(* CODESYS project IoDrvMasterTemplateIEC.library
   Author: 3S - Smart Software Solutions GmbH
   Title: IoDrvMasterTemplateIEC
   Version: 3.5.15.0
   Placeholder: PlaceholderTemplate
   DocFormat: reStructuredText
   Company: MyCompany
   LanguageModelAttribute: qualified-access-only
   DefaultNamespace: TMP

Project tree, tasks and I/O mapping:
  libraries: SysMem, * (System); SysCpuHandling, * (System); IoDrvBase, * (System); IoDriver Parameter Interfaces, * (System); Base Interfaces, * (System); IoDriver Interfaces, * (System); CmpErrors2 Interfaces, * (System); SysTypes2 Interfaces, * (System); CAA Device Diagnosis, * (CAA Technical Workgroup); CAA Types Extern, * (CAA Technical Workgroup); CmpAsyncMgr, * (System); Network, 3.5.7.0 (3S - Smart Software Solutions GmbH); IoStandard, 3.5.13.0 (System); IoDrvUtility, 3.5.15.0 (3S - Smart Software Solutions GmbH); SysSem, * (System)
  00000000-0000-0000-0000-000000000000|D:\CoDeSys\LibrariesV3\trunk\Intern\CAA\CAA Template\3.2.0.3 draft\Prefix.pdf
  00000000-0000-0000-0000-000000000000|D:\CoDeSys\LibrariesV3\trunk\Intern\CAA\CAA Template\3.4.0.0 draft\Placeholder.xml
  00000000-0000-0000-0000-000000000000|D:\CoDeSys\LibrariesV3\trunk\Intern\CAA\CAA Template\3.5.2.0 draft\Placeholder.xml
  IoDrvMasterTemplateIEC/
    Enums/
      data type IoType
    Function Blocks/
      function block FixedArrayList [ST]: Create, Destroy, Get, Size
      function block IoDrvTemplateMaster [ST]: IoDrvReadInputs, IoDrvIdentify, IoDrvUpdateConfiguration, IoDrvWatchdogTrigger, IoDrvScanModules, IoDrvUpdateMapping, IoDrvWriteOutputs, IoDrvStartBusCycle, IoDrvGetModuleDiagnosis, IoDrvWriteParameter, IoDrvReadParameter, QueryInterface, FB_Reinit, Initialize, FB_Exit, FB_Init, IoDrvGetConnector, Cleanup, FreeScanData
      function block IoDrvTemplateModule [ST]: Initialize, UpdateConfigurationCreate, UpdateConfigurationDestroy, StartBusCycle, ModuleID, IsDisabled
      function block IoDrvTemplateSlave [ST]: Initialize, UpdateConfigurationCreate, UpdateConfigurationDestroy, StartBusCycle, SlaveID, IsDisabled
      function block IoDrvTemplateMasterDiag [ST]: ChildNodeCount, Connector, Enable, FirstChildNode, Index, IsRootNode, NextSiblingNode, ParentNode, SiblingNodeCount, GetChild, Initialize_Diag, GetSpecificDeviceState, SetCommunicationState, GetDeviceInfo, GetDeviceErrorAsync, GetSpecificDeviceErrorAsync, GetDeviceDiagnosisInfo, GetDeviceState, CheckCurrentSupportedCommunicationState, CheckSupportedCommunicationState, GetQoS, GetBusErrorAsync, GetBusDiagnosisInfo, GetBusState, GetBusInfo, GetSpecificBusState, GetLogger, GetBusScanAsync, ReconfigureActive, SiblingIRP, ReconfigureAsync, RegisterIRPChild
      function block IoDrvTemplateSlaveDiag [ST]: ChildNodeCount, Connector, Enable, FirstChildNode, Index, IsRootNode, NextSiblingNode, ParentNode, SiblingNodeCount, GetChild, Initialize_Diag, GetSpecificDeviceState, SetCommunicationState, GetDeviceInfo, GetDeviceErrorAsync, GetSpecificDeviceErrorAsync, GetDeviceDiagnosisInfo, GetDeviceState, CheckCurrentSupportedCommunicationState, CheckSupportedCommunicationState, GetQoS, GetBusErrorAsync, GetBusDiagnosisInfo, GetBusState, GetBusInfo, GetSpecificBusState
      function block IoDrvTemplateModuleDiag [ST]: ChildNodeCount, Connector, Enable, FirstChildNode, Index, IsRootNode, NextSiblingNode, ParentNode, SiblingNodeCount, GetChild, Initialize_Diag, GetSpecificDeviceState, SetCommunicationState, GetDeviceInfo, GetDeviceErrorAsync, GetSpecificDeviceErrorAsync, GetDeviceDiagnosisInfo, GetDeviceState, CheckCurrentSupportedCommunicationState, CheckSupportedCommunicationState, GetQoS, GetBusErrorAsync, GetBusDiagnosisInfo, GetBusState, GetBusInfo, GetSpecificBusState
    GlobalConstants/
      global variables PARAMS_IODRVTEMPLATEMASTER
    Structs/
      data type IoEntry
      data type Module
      data type Slave
      data type UdpIO
    _ExternalFilesDoku/
      M_AblaufProto
      M_Behave
      M_Connectors
      M_cycle
      M_Proto
      M_Tree
      M_run
  00000000-0000-0000-0000-000000000000|D:\CODESYS\CodesysSpV3\CodesysSpV3\Templates\IoDrvMasterTemplateIEC\RestoreOld\DokPic\M_AblaufProto.png
  00000000-0000-0000-0000-000000000000|D:\CODESYS\CodesysSpV3\CodesysSpV3\Templates\IoDrvMasterTemplateIEC\RestoreOld\DokPic\M_Behave.png
  00000000-0000-0000-0000-000000000000|D:\CODESYS\CodesysSpV3\CodesysSpV3\Templates\IoDrvMasterTemplateIEC\RestoreOld\DokPic\M_Connectors.png
  00000000-0000-0000-0000-000000000000|D:\CODESYS\CodesysSpV3\CodesysSpV3\Templates\IoDrvMasterTemplateIEC\RestoreOld\DokPic\M_cycle.png
  00000000-0000-0000-0000-000000000000|D:\CODESYS\CodesysSpV3\CodesysSpV3\Templates\IoDrvMasterTemplateIEC\RestoreOld\DokPic\M_Proto.png
  00000000-0000-0000-0000-000000000000|D:\CODESYS\CodesysSpV3\CodesysSpV3\Templates\IoDrvMasterTemplateIEC\RestoreOld\DokPic\M_Tree.png
  00000000-0000-0000-0000-000000000000|D:\CODESYS\CodesysSpV3\CodesysSpV3\Templates\IoDrvMasterTemplateIEC\RestoreOld\DokPic\M_run.png
*)

// IoDrvMasterTemplateIEC/Structs/IoEntry
/// Is generated for each output and input, when an ouput or input exsits in the Slave (type 3) or modules(all types).
/// This saves time in ``IoDrvTemplateMaster.IoDrvStartBusCycle``, because iterating over the ConnectorList and searching for the out- and inputs takes time. This is done in ''IoDrvTemplateMaster.IoDrvUpdateConfiguration'', where a fixed arrayList is generated. 
TYPE IoEntry :
STRUCT
    /// Input or output?
	ioType: IoType;
    /// Pointer to the Parameter. 
	pParameter: POINTER TO IoConfigParameter;
END_STRUCT
END_TYPE

// IoDrvMasterTemplateIEC/Structs/Module
/// This struct is generated, for each Module in the device tree in the ''IoDrvTemplateSlave'' FB, to access the Slaves over a pointer an not over the ConenctorList. This saves time in the ''IoDrvTemplateMaster.IoDrvStartBusCycle'' method. 
TYPE Module :
STRUCT
	moduleInstance : POINTER TO IoDrvTemplateModule;		
END_STRUCT
END_TYPE

// IoDrvMasterTemplateIEC/Structs/Slave
/// This struct is generated, for each Slave in the device tree in the ''IoDrvTemplateMaster'' FB, to access the Slaves over a pointer an not over the ConenctorList. This saves time in the ''IoDrvTemplateMaster.IoDrvStartBusCycle'' method. 
TYPE Slave :
STRUCT
	slaveInstance : POINTER TO IoDrvTemplateSlave;		
END_STRUCT
END_TYPE

// IoDrvMasterTemplateIEC/Structs/UdpIO
/// Information, which are needed also in the modules an slaves. This struct function is to bundle this information and pass them down in the stack easily. 
TYPE UdpIO :
STRUCT
	r_udpInBuffer: POINTER TO FixedArrayList;
	r_BytesReceived : CAA.SIZE;

	s_udpSender : POINTER TO NBS.UDP_Send;
	s_udpPeer: POINTER TO NBS.UDP_Peer ;
	s_portSendTo : UINT;
	s_ipSendTo : POINTER TO NBS.IP_ADDR;
	s_udpOutBuffer: POINTER TO FixedArrayList;	
END_STRUCT
END_TYPE

// IoDrvMasterTemplateIEC/Enums/IoType
{attribute 'qualified_only'}
{attribute 'strict'}
/// Used in |IoEntry|.
TYPE IoType :
(
	INPUT := 0,
	OUTPUT := 1
);
END_TYPE

// IoDrvMasterTemplateIEC/GlobalConstants/PARAMS_IODRVTEMPLATEMASTER
VAR_GLOBAL
	/// This string is used, when memory is allocated. 
    g_stComponentName : STRING := 'IoDrvMasterTemplate';
	
	/// The ID at which the ParameterId for the inputs start in the deviceDescription (xml-file). This is a running nummer. The loop stops, if there is an unused number: 2000, 2001, 2002, 2004 --> after 2002 no entries would be processed.
	START_OF_INPUTPARAMS : UDINT := 2000;
   
	/// The ID at which the ParameterId for the inputs end in the deviceDescription (xml-file).
	END_OF_INPUTPARAMS : UDINT := 2999;

    /// Same as for inputs. 	
	START_OF_OUTPUTPARAMS : UDINT := 3000;
    /// Same as for inputs. 
	END_OF_OUTPUTPARAMS : UDINT := 3999;

    /// The size of the UDP-Buffer to send messages.  
	SIZE_OF_INPUT_OUTPUT_BUFFER : UDINT := 30;
	
END_VAR

// IoDrvMasterTemplateIEC/Function Blocks/FixedArrayList
(*
 .. code-block:: codesys
  
    VAR_GLOBAL CONSTANT
        g_stComponentName : STRING := 'MyApp';
    END_VAR
    
    TYPE MyStruct:
    STRUCT
        someData1: DWORD;
        someData2: BYTE;
    END_STRUCT
    END_TYPE
    
    _fixedArrayList :FixedArrayList
    pMyStruct : POINTER TO MyStruct;
    numberOfEntries: DWORD;
    
    numberOfEntries := 10;
    IF( NOT _fixedArrayList(numberOfEntries, SIZEOF(MyStruct:), g_stComponentName) ) THEN 
        RETURN; //error no free space ....
    END_IF
    
	IF _fixedArrayList.Size > 0 THEN
		FOR i:=0 TO _fixedArrayList.Size - 1 DO
			pMyStruct := _fixedArrayList.Get(i);
			// do something ...			
		END_FOR
	END_IF
*)
FUNCTION_BLOCK FixedArrayList
VAR_INPUT
END_VAR
VAR_OUTPUT
END_VAR
VAR
    /// Address to the memblock. 
	_varMem: POINTER TO BYTE := 0;
    /// How many entries.
	_sizeOfArray: DWORD;
    /// Given in Create.
	_sizeOfObjectInByte: DWORD;
    /// Needed by Destroy
	_stComponentName: STRING;
END_VAR

/// Creates a fixed memmory block, which can be accessed over an index.
METHOD Create : BOOL
VAR_INPUT
    /// How many entries should be available?
	sizeOfArray: DWORD;
    /// How big in bytes is one entry?
	sizeOfObjectInByte: DWORD;
    /// Which component is using this memory? If the memory is not freed after shutdown, a warning with this string is generated.
	stComponentName : STRING;
END_VAR

VAR
	iecResult : RTS_IEC_Result;
END_VAR
_sizeOfArray := sizeOfArray;
_sizeOfObjectInByte := sizeOfObjectInByte;
_stComponentName := stComponentName;
_varMem :=  SysMemAllocData(_stComponentName, _sizeOfObjectInByte*_sizeOfArray , ADR(iecResult));


Create := (iecResult = CmpErrors.Errors.ERR_OK); // if false -> _varMem=0 (impicit)
END_METHOD

/// Frees the memory, which was allocated in |FixedArrayList.Create|, if it was successful.
METHOD Destroy
VAR_INPUT
END_VAR
IF(_varMem <> 0) THEN
	SysMemFreeData(_stComponentName, _varMem);
END_IF
END_METHOD

/// Returns a pointer to the element at the given index.
/// :return: The address to the element, if the index is valid, else 0.
METHOD Get : POINTER TO BYTE
VAR_INPUT
    /// Index of the element, which should be accessed. The index is between 0 and DWORD.maxValue.
	index: DWORD;
END_VAR
IF( index < _sizeOfArray) THEN
	Get := (_varMem + _sizeOfObjectInByte*index);
ELSE
	Get := 0;
END_IF
END_METHOD

/// Reads the amount of elements, which can be accessed. Is for the use in loops to iterate over all elements. 
PROPERTY Size : DWORD
GET
Size := _sizeOfArray;
END_GET
END_PROPERTY

END_FUNCTION_BLOCK

// IoDrvMasterTemplateIEC/Function Blocks/IoDrvTemplateMaster
{attribute 'no_assign'}
{attribute 'conditionalshow_all_locals' := 'IoDrvDebug'}
FUNCTION_BLOCK IoDrvTemplateMaster EXTENDS IoDrvBase IMPLEMENTS ICmpIoDrvParameter
VAR_INPUT
END_VAR
VAR_OUTPUT
END_VAR
VAR CONSTANT
	CLASSID_CCmpIoDrvTemplate : DWORD := 16#0000FF02;
END_VAR
VAR
	_IIoDrv : ICmpIoDrv;
	_IIoDrvParameter : ICmpIoDrvParameter;
	
	_xBackGroundDiagStarted : BOOL;
	_bDeactivated : BOOL;

    // used to save the slaves with their slaveID in a list. To access the correct slave in the method IoDrvStartBusCylce fast.  
	_fal_shortcut2Slaves :FixedArrayList; 
	
	//Variables for scan
	_iScannedSlaves : INT;
	_pScanList : POINTER TO IoStandard.IoConfigConnector;

    // UDP server varaibles
	_udpPeer: NBS.UDP_Peer ;
	_iPAddr :  NBS.IP_ADDR;
	_uiPortReceive : UINT;
	_udpRec : NBS.UDP_Receive;
	_udpSend : NBS.UDP_Send;
	_udpInBuffer, _udpOutBuffer: FixedArrayList;

	_myState: BYTE := 1; // remember the state
	_connectorFlagController: IoDrvUtility.ConnectorFlagController;
	
//	_lock: RTS_IEC_Handle;
END_VAR

{attribute 'conditionalshow' := 'IoDrvDebug'}
METHOD IoDrvReadInputs : UDINT
VAR_INPUT
	pConnectorMapList : POINTER TO IoConfigConnectorMap;
	nCount : DINT;
END_VAR
VAR
	i,j : DINT;
	pConnectorMap : POINTER TO IoStandard.IoConfigConnectorMap;
	pChannelMap : POINTER TO IoStandard.IoConfigChannelMap;
END_VAR
IoDrvReadInputs_Count := IoDrvReadInputs_Count + 1;

IF pConnectorMapList = 0 OR nCount = 0 THEN
	IoDrvReadInputs := Errors.ERR_PARAMETER;
	RETURN;
END_IF

FOR i:=0 TO nCount - 1 DO
	pConnectorMap := ADR(pConnectorMapList[i]);
	
	FOR j:= 0 TO UDINT_TO_UINT(pConnectorMap^.dwNumOfChannels) - 1 DO
		pChannelMap := ADR(pConnectorMap^.pChannelMapList[j]);
		
		// input medium byteorder: Little Endian:		
		IoMgrCopyInputLE(pChannelMap, pChannelMap^.pParameter^.dwDriverSpecific);
		
		// input medium byteorder: Big Endian:		
		//IoMgrCopyInputBE(ADR(pChannelMap, pChannelMap^.pParameter^.dwDriverSpecific);
	END_FOR
END_FOR

IoDrvReadInputs := Errors.ERR_OK;
END_METHOD

{attribute 'conditionalshow' := 'IoDrvDebug'}
METHOD IoDrvIdentify : UDINT
VAR_INPUT
	pConnector : POINTER TO IoConfigConnector;	
END_VAR
VAR
END_VAR
IoDrvIdentify_Count := IoDrvIdentify_Count + 1;
IoDrvIdentify := Errors.ERR_NOTIMPLEMENTED;
END_METHOD

{attribute 'conditionalshow' := 'IoDrvDebug'}
METHOD IoDrvUpdateConfiguration : UDINT
VAR_INPUT
	pConnectorList : POINTER TO IoConfigConnector;
	nCount : DINT;
END_VAR
VAR
	p_dwParValueSlave : POINTER TO IoDrvTemplateSlave;
	pParameter : POINTER TO IoConfigParameter;	
	pDummy			: POINTER TO XWORD;
	
	pChild : POINTER TO IoConfigConnector;	
	pstConnectorVendorName : POINTER TO STRING;
	pstConnectorDeviceName : POINTER TO STRING;
	dwTest,i : DWORD;
	Result : UDINT := 0;
	xDisabled : BOOL;
	
	slaveCount : UDINT := 0;
	slaveIter : POINTER TO Slave;
	
	nCountRemember: DINT;
	
	pstDummy : POINTER TO STRING;
END_VAR
IoDrvUpdateConfiguration_Count := IoDrvUpdateConfiguration_Count + 1;
IoDrvUpdateConfiguration := Errors.ERR_OK;

IF pConnectorList = 0 THEN // destroy -> time to clean up
	// Reset application
	m_pConnector^.hIoDrv := 0; 
	m_pConnector^.pFather^.hIoDrv := 0;
	
	Cleanup();
	_udpOutBuffer.Destroy();
	_udpInBuffer.Destroy();
	//Go through all childs of the device
	IF _fal_shortcut2Slaves.Size > 0 THEN
		FOR i:=0 TO _fal_shortcut2Slaves.Size - 1 DO
			slaveIter := _fal_shortcut2Slaves.Get(i);
			slaveIter^.slaveInstance^.UpdateConfigurationDestroy(); // childs of master are IoDrvTemplateSlave FB´s -> call UpdateConfigurationDestroy(...) to give them the chance to cleanup
		END_FOR
	END_IF
	_fal_shortcut2Slaves.Destroy();// delete shortcut list to slaves 	

	// reset var´s (needed when reconfigure is activated)
	_iScannedSlaves := 0;
	_pScanList := 0;
	_myState := 1; // remember the state
	
	RETURN; // nothing more to do
END_IF

m_pConnector := IoMgrConfigGetConnector(pConnectorList, ADR(nCount), m_wModuleType, m_dwInstance);
nCountRemember := nCount; // to reset the counter to iterate over the childs
_connectorFlagController.Init(m_pConnector, nCount, FALSE); // ^.pFather is MasterIECDriver::Connector::256
_connectorFlagController.AutoSetErrorClearedFlag := TRUE; //use the generic algorithm for setting the Error Cleared flag in device tree.
_connectorFlagController.DiagProvider := TRUE;

IF m_pConnector = 0 THEN
	IoDrvUpdateConfiguration := ERRORS.ERR_PARAMETER;
	RETURN;
END_IF

//check if device is enabled in the device tree
_bDeactivated := _connectorFlagController.State = IoDrvUtility.ConnectorState.DISABLED;

IF _bDeactivated THEN // IO changes don´t care, if device is disabled.
	m_pConnector^.hIoDrv := 0;
	m_pConnector^.pFather^.hIoDrv := 0;
	IoDrvUpdateConfiguration := CmpErrors.Errors.ERR_OK;
	RETURN;
END_IF

IF (m_pConnector^.hIoDrv = 0) and (NOT _bDeactivated) THEN // register to get called, when IO changed
	m_pConnector^.hIoDrv := m_hInterface; 
	m_pConnector^.pFather^.hIoDrv := m_hInterface;
END_IF

IF m_pConnector^.hIoDrv = m_hInterface THEN
	{IF defined (pou:IoMgrSetDriverProperties)}			
		IoMgrSetDriverProperties(m_hInterface, DRVPROP_CONSISTENCY OR DRVPROP_BACKGROUND_GETDIAG);
		//Note: background diagnosis property flag is optional (supported with 3.5.1.0 runtime)
	{END_IF}										

	//Read some parameters
	pParameter := IoMgrConfigGetParameter(m_pConnector, 393218);
	IF pParameter <> 0 THEN
		pstConnectorVendorName := IoMgrConfigGetParameterValuePointer(pParameter, ADR(Result));
	END_IF
	pParameter := IoMgrConfigGetParameter(m_pConnector, 393219);
	IF pParameter <> 0 THEN
		pstConnectorDeviceName := IoMgrConfigGetParameterValuePointer(pParameter, ADR(Result));
	END_IF
	pParameter := IoMgrConfigGetParameter(m_pConnector, 393220);	(* test parameter *)
	IF (pParameter <> 0) THEN
		dwTest := IoMgrConfigGetParameterValueDword(pParameter, ADR(Result));	(* Test parameter value *)			
	END_IF
	
	pParameter := IoMgrConfigGetParameter(m_pConnector, 256);	// ip addr
	IF (pParameter <> 0) THEN
		pstDummy := IoMgrConfigGetParameterValuePointer(pParameter, ADR(Result));
		_iPAddr.sAddr := pstDummy^;
	END_IF
	
	pParameter := IoMgrConfigGetParameter(m_pConnector, 257);	// port
	IF (pParameter <> 0) THEN
		_uiPortReceive := DWORD_TO_UINT( IoMgrConfigGetParameterValueWord (pParameter, ADR(Result)) );		
	END_IF

	
	//Go through all childs of the device
	nCount:= nCountRemember;
	slaveCount :=0; // save amount of slaves
	pChild := IoMgrConfigGetFirstChild(m_pConnector, ADR(nCount), m_pConnector);
	WHILE (pChild <> 0) DO
		// childs of master are IoDrvTemplateSlave FB´s -> call UpdateConfigurationCreate(...) to let them init()
		pParameter := IoMgrConfigGetParameter(pChild, 1); 
		IF pParameter <> 0 THEN
			pDummy := ConfigGetParameterValuePointer(pParameter,ADR(Result));
			p_dwParValueSlave :=  pDummy^;
			IF p_dwParValueSlave <> 0 THEN
				p_dwParValueSlave^.UpdateConfigurationCreate(pConnector := pChild, m_hInterface, nCount, xDisabled => xDisabled);
				IF NOT xDisabled THEN
					slaveCount := slaveCount + 1;
				END_IF
			END_IF
		END_IF

		pChild := IoMgrConfigGetNextChild(pChild, ADR(nCount), m_pConnector);
	END_WHILE
	
	// save a shortcut to know which IoDrvTemplateSlave instance is in resposable to which slaveID and save this in a variable memory block (_fal_shortcut2Slaves) to access it without going over the slowly connectorList (IoMgrConfigGetFirstChild) 
	// this _fal_shortcut2Slaves is needed in the IoDrvStartBusCycle method to be fast
	IF( NOT _fal_shortcut2Slaves.Create( slaveCount, SIZEOF(Slave), g_stComponentName) ) THEN
		IoDrvUpdateConfiguration := Errors.ERR_FAILED; // no space ....
		RETURN;
	END_IF
	
	nCount:= nCountRemember;
	pChild := IoMgrConfigGetFirstChild(m_pConnector, ADR(nCount), m_pConnector);
	i := 0;
	WHILE (pChild <> 0) DO
		pParameter := IoMgrConfigGetParameter(pChild, 1); 
		IF pParameter <> 0 THEN
			pDummy := ConfigGetParameterValuePointer(pParameter,ADR(Result));
			p_dwParValueSlave :=  pDummy^;
			IF p_dwParValueSlave <> 0 THEN
				IF NOT p_dwParValueSlave^.IsDisabled THEN
					slaveIter := _fal_shortcut2Slaves.Get(i); // get next place to save the slaveInstance
					i := i + 1;
					slaveIter^.slaveInstance := p_dwParValueSlave;
				END_IF
			END_IF
		END_IF
		pChild := IoMgrConfigGetNextChild(pChild, ADR(nCount), m_pConnector);
	END_WHILE

	_connectorFlagController.State := IoDrvUtility.ConnectorState.RUNNING;
END_IF
END_METHOD

{attribute 'conditionalshow' := 'IoDrvDebug'}
METHOD IoDrvWatchdogTrigger : UDINT
VAR_INPUT
	pConnector : POINTER TO IoConfigConnector;	
END_VAR
VAR
END_VAR
IoDrvWatchdogTrigger_Count := IoDrvWatchdogTrigger_Count + 1;
IoDrvWatchdogTrigger := Errors.ERR_OK;
END_METHOD

{attribute 'conditionalshow' := 'IoDrvDebug'}
METHOD IoDrvScanModules : UDINT
VAR_INPUT
	pConnector : POINTER TO IoConfigConnector;
	ppConnectorList : POINTER TO POINTER TO IoConfigConnector;
	pnCount : POINTER TO DINT;	
END_VAR
VAR
	pCurConnector : POINTER TO IoConfigConnector;
	pParameter: POINTER TO IoConfigParameter;
	pString : POINTER TO STRING;
	i : INT;
END_VAR
IoDrvScanModules_Count := IoDrvScanModules_Count + 1;

IF pConnector = 0 OR ppConnectorList = 0 OR pnCount = 0 THEN
	IoDrvScanModules := Errors.ERR_PARAMETER;
	RETURN;
END_IF

FreeScanData();

pnCount^ := 0;
ppConnectorList^ := 0;

(*
	TODO: implement specific bus scan!
	Note: IoDrvScanModules is called in communication task. If this method takes too long (> 20s) a communication timeout may happen.
	In this cases you can do a segmented scan by setting IoStandard.ConnectorOptions.CO_SCAN_PENDING_SUPPORTED.
	If IoDrvScanModules returns ERR_PENDING method is called again. The results of all calls are combined by the GUI.
*)

(*The following code just generates some example data. The real scan algorithm has to set the values regarding to the scan result. *)
_iScannedSlaves := 2; //we return 2 slaves

IF _iScannedSlaves > 0 THEN
	//Allocate memory for the connector list
	ppConnectorList^ := SysMemAllocData(g_stComponentName, UINT_TO_DWORD(INT_TO_UINT(_iScannedSlaves) * SIZEOF(IoStandard.IoConfigConnector)), 0);
	IF ppConnectorList = 0 THEN
		IoDrvScanModules := Errors.ERR_FAILED;
		_iScannedSlaves := 0;
		RETURN;
	END_IF
	SysMem.SysMemSet(ppConnectorList^, 0, UINT_TO_DWORD(INT_TO_UINT(_iScannedSlaves) * SIZEOF(IoStandard.IoConfigConnector)));
END_IF

pCurConnector := ppConnectorList^;
FOR i := 0 TO _iScannedSlaves - 1 DO
	pCurConnector^.dwNumOfParameters := 4; //we return the 4 mandatory parameters
	//Alocate memory for the parameter list of the current connector
	pCurConnector^.pParameterList := SysMemAllocData(g_stComponentName, pCurConnector^.dwNumOfParameters * SIZEOF(IoStandard.IoConfigParameter), 0);
	SysMem.SysMemSet(pCurConnector^.pParameterList, 0, pCurConnector^.dwNumOfParameters * SIZEOF(IoStandard.IoConfigParameter));
	
    pParameter := pCurConnector^.pParameterList;
	
	//Set parameter: Vendor code
	pParameter^.dwParameterId := 1;
	pParameter^.dwValue := 1; //Vendor Code
	pParameter^.wLen := 32;
	pParameter^.wType := INT_TO_WORD(TypeClass.TYPE_DWORD); //16#4
	pParameter^.dwFlags := IoStandard.PVF_READ OR IoStandard.PVF_WRITE OR IoStandard.PVF_VALUE; //16#34
	
	pParameter := pParameter + SIZEOF(IoStandard.IoConfigParameter);
	
	//Set parameter: Product code
	pParameter^.dwParameterId := 2;
	pParameter^.dwValue := 2; //Product Code
	pParameter^.wLen := 32;
	pParameter^.wType := INT_TO_WORD(TypeClass.TYPE_DWORD); //16#4
	pParameter^.dwFlags := IoStandard.PVF_READ OR IoStandard.PVF_WRITE OR IoStandard.PVF_VALUE; //16#34
	
	pParameter := pParameter + SIZEOF(IoStandard.IoConfigParameter);
	
	//Set parameter: Revision Number
	pParameter^.dwParameterId := 3;
	pParameter^.dwValue :=3; //Revision Number
	pParameter^.wLen := 32;
	pParameter^.wType := INT_TO_WORD(TypeClass.TYPE_DWORD); //16#4
	pParameter^.dwFlags := IoStandard.PVF_READ OR IoStandard.PVF_WRITE OR IoStandard.PVF_VALUE; //16#34
	
	pParameter := pParameter + SIZEOF(IoStandard.IoConfigParameter);
	
	
	(* Slave_T1_IECDriver.xml:
	
			<DeviceIdentification>
				<Type>40102</Type>
				<Id>1001 0001</Id>
	*)		
			
	//Set parameter: Device Identification
	pParameter^.dwParameterId := 4;
	pParameter^.dwValue := SysMemAllocData(g_stComponentName, SIZEOF(STRING), 0);
	pString := pParameter^.dwValue;
	pString^ := '1001 0001'; // Device Identification <Id>1001 0001</Id>
	pParameter^.wLen := SIZEOF(STRING);
	pParameter^.wType := INT_TO_WORD(TypeClass.TYPE_STRING); //16#10
	pParameter^.dwFlags := IoStandard.PVF_READ OR IoStandard.PVF_WRITE OR IoStandard.PVF_POINTER; //16#32
		
	pCurConnector^.hIoDrv := THIS;
	pCurConnector^.pFather := pConnector;
	pCurConnector^.wType := 40102; // <Type>40102</Type>
	
	pCurConnector := pCurConnector + SIZEOF(IoStandard.IoConfigConnector);
END_FOR

pnCount^ := _iScannedSlaves; //Set number of scanned devices
IoDrvScanModules := CmpErrors.Errors.ERR_OK;
END_METHOD

{attribute 'conditionalshow' := 'IoDrvDebug'}
METHOD IoDrvUpdateMapping : UDINT
VAR_INPUT
	pTaskMapList : POINTER TO IoConfigTaskMap;
	nCount : DINT;	
END_VAR
VAR
END_VAR
IoDrvUpdateMapping_Count := IoDrvUpdateMapping_Count + 1;

IF (pTaskMapList = 0) THEN
	IoDrvUpdateMapping := Errors.ERR_PARAMETER;
	RETURN;
END_IF

IoDrvUpdateMapping := Errors.ERR_OK;
END_METHOD

{attribute 'conditionalshow' := 'IoDrvDebug'}
METHOD IoDrvWriteOutputs : UDINT
VAR_INPUT
	pConnectorMapList : POINTER TO IoConfigConnectorMap;
	nCount : DINT;
END_VAR
VAR
	i,j : DINT;
	pConnectorMap : POINTER TO IoStandard.IoConfigConnectorMap;
	pChannelMap : POINTER TO IoStandard.IoConfigChannelMap;
END_VAR
IoDrvWriteOutputs_Count := IoDrvWriteOutputs_Count + 1;

IF pConnectorMapList = 0 OR nCount = 0 THEN
	IoDrvWriteOutputs := Errors.ERR_PARAMETER;
	RETURN;
END_IF

FOR i:=0 TO nCount - 1 DO
	pConnectorMap := ADR(pConnectorMapList[i]);
	
	FOR j:= 0 TO UDINT_TO_UINT(pConnectorMap^.dwNumOfChannels) - 1 DO
		pChannelMap := ADR(pConnectorMap^.pChannelMapList[j]);
		
		// output medium byteorder: Little Endian:		
		IoMgrCopyOutputLE(pChannelMap, pChannelMap^.pParameter^.dwDriverSpecific);
		
		// output medium byteorder: Big Endian:		
		//IoMgrCopyOutputBE(pChannelMap, pChannelMap^.pParameter^.dwDriverSpecific);
	END_FOR
END_FOR

IoDrvWriteOutputs := Errors.ERR_OK;
END_METHOD

{attribute 'conditionalshow' := 'IoDrvDebug'}
METHOD IoDrvStartBusCycle : UDINT
VAR_INPUT
	pConnector : POINTER TO IoConfigConnector;
END_VAR
VAR
	i : DWORD;
	slaveIter : POINTER TO Slave;
	udpIo: UdpIO;
	ipMulti :  NBS.IP_ADDR;
END_VAR
IoDrvStartBusCycle_Count := IoDrvStartBusCycle_Count + 1;

IF _bDeactivated OR_ELSE pConnector <> m_pConnector THEN
	RETURN;
END_IF

//if background diagnosis is not active call IoDrvGetModuleDiagnosis; normally it will be called by the runtime if DRVPROP_BACKGROUND_GETDIAG is set
IF NOT _xBackGroundDiagStarted THEN
	IoDrvGetModuleDiagnosis(m_pConnector); //DRVPROP_BACKGROUND_GETDIAG not set or runtime version < V3.5.1.0
END_IF

//optional: call IoDrvWatchdogTrigger or set driver property DRVPROP_WATCHDOG in UpdateConfiguration
IoDrvWatchdogTrigger(pConnector);

//	---------------------------------------------------------------------------------------
//  Here is the place for your statemachine to realize the communication over the bussystem
//  ---------------------------------------------------------------------------------------
CASE _myState OF
	1: // init
		ipMulti.sAddr := '';
		_udpPeer(xEnable := TRUE, ipAddr := _iPAddr, uiPort := _uiPortReceive, ipMultiCast := ipMulti );
		IF _udpPeer.xBusy AND _udpPeer.hPeer <> CAA.gc_hINVALID AND _udpInBuffer.Create(SIZE_OF_INPUT_OUTPUT_BUFFER, SIZEOF(BYTE), g_stComponentName) 
					AND _udpOutBuffer.Create(SIZE_OF_INPUT_OUTPUT_BUFFER, SIZEOF(BYTE), g_stComponentName) 
			THEN
			_myState := 2;
		ELSE
			_myState :=99;
		END_IF
	2: // running
		// read inputs, response to read outputs request
		REPEAT
			_udpRec(xEnable := TRUE, hPeer :=  _udpPeer.hPeer, szSize := SIZE_OF_INPUT_OUTPUT_BUFFER, pData := _udpInBuffer.Get(0));
			
			//_udpSend(xExecute := TRUE, udiTimeOut := 0, hPeer := _udpPeer, ipAddr := _udpRec.ipFrom, uiPort := _uiPortSend, szSize := 3, pData := _udpOutBuffer);
						
			IF _udpRec.szCount > 0 THEN
				// in the first byte is the slaveID -> search the slave with this id and call the instance
				IF _fal_shortcut2Slaves.Size > 0 THEN
					FOR i:=0 TO _fal_shortcut2Slaves.Size - 1 DO
						slaveIter := _fal_shortcut2Slaves.Get(i);
						IF(_udpRec.szSize > 0) THEN
							IF( slaveIter^.slaveInstance^.SlaveID = _udpInBuffer.Get(0)^ ) THEN // slaveId received (first byte) = slaveId of the instance?
								// bundle information of receive and infos to answere on a request together 
								udpIo.r_udpInBuffer := ADR(_udpInBuffer);
								udpIo.r_BytesReceived := _udpRec.szCount;
								udpIo.s_udpSender := ADR(_udpSend);
								udpIo.s_udpPeer	 := ADR(_udpPeer);
								udpIo.s_portSendTo := _udpRec.uiPortFrom;
								udpIo.s_ipSendTo := ADR(_udpRec.ipFrom);
								udpIo.s_udpOutBuffer := ADR(_udpOutBuffer);
								
								slaveIter^.slaveInstance^.StartBusCycle(udpIo); // call by ref. ...
							END_IF
						END_IF
					END_FOR
				END_IF
			END_IF
		UNTIL
			NOT _udpRec.xReady
		END_REPEAT

		IF _fal_shortcut2Slaves.Size > 0 THEN
			FOR i:=0 TO _fal_shortcut2Slaves.Size - 1 DO // call all slaves with type= 3 -> no communication only linking in to outputs...
				slaveIter := _fal_shortcut2Slaves.Get(i);
				IF( slaveIter^.slaveInstance^.SlaveID = 3) THEN
					slaveIter^.slaveInstance^.StartBusCycle(udpIo); // udpIo is dummy, is not used by type 3
				END_IF
			END_FOR
		END_IF
		// search the slave, who is resposable for the message (first byte is 
	99: // error
		;
END_CASE

	//Go through all childs of the device

IoDrvStartBusCycle := Errors.ERR_OK;
END_METHOD

METHOD IoDrvGetModuleDiagnosis : UDINT
VAR_INPUT
	pConnector : POINTER TO IoConfigConnector;
END_VAR
VAR
END_VAR
IF pConnector = 0 THEN
	//we are called from the background task
	_xBackGroundDiagStarted := TRUE;
END_IF

// update connectorflags if something changed -> here depending on your state of your driver set when e.g. running to: _scf.State := IoDrvUtility.ConnectorState._scf.State := IoDrvUtility.ConnectorState.RUNNING; 
// This will update the dwFlags of the Connector and depending on them the icon in front of the device will change (read doku of IoDrvUtility)

IoDrvGetModuleDiagnosis_Count := IoDrvGetModuleDiagnosis_Count + 1;
IoDrvGetModuleDiagnosis := Errors.ERR_NOTIMPLEMENTED;
END_METHOD

{attribute 'conditionalshow' := 'IoDrvDebug'}
METHOD IoDrvWriteParameter : UDINT
VAR_INPUT
	pConnector : POINTER TO IoConfigConnector;
	pParameter : POINTER TO IoConfigParameter;
	pData : POINTER TO BYTE;
	dwBitSize : DWORD;
	dwBitOffset : DWORD;
END_VAR
VAR
	pParam : POINTER TO IoConfigParameter;
	pstDiagString : POINTER TO STRING;
	pValue : POINTER TO BYTE;
END_VAR
IF pConnector = 0 OR pParameter = 0 OR pData = 0 THEN
	IoDrvWriteParameter := Errors.ERR_PARAMETER;
	RETURN;	
END_IF

//If IoDrvWriteParameter returns a value unequal ERR_OK, write parameter will be handled by the IO-manager!
//Note: Code must be only implemented here if there are special things to do.

IoDrvWriteParameter := Errors.ERR_OK;

CASE pParameter^.dwParameterId OF
	393221: //simulate diag
		IF pData^ <> 0 THEN
			(*
				Example for extended Diagnostic:
				- here a string value is written to parameter of channeltype "diag": when "CF_CONNECTOR_DIAGNOSTIC_AVAILABLE" is set in the connector, the diagnostic message is read with ReadParameter.
			*)
			pParam := IoMgrConfigGetParameter(pConnector, 4711);
			IF pParam <> 0 THEN
				pstDiagString := IoMgrConfigGetParameterValuePointer(pParam, 0);
				IF pstDiagString <> 0 THEN
					pstDiagString^ := 'Error pending';
				END_IF
			END_IF
			
			(*
				set diagnostic available flag to trigger reading of diagnosis parameter
			*) 
			IoMgrConfigSetDiagnosis(pConnector, Connectorflags.CF_CONNECTOR_DIAGNOSTIC_AVAILABLE);
		END_IF
		RETURN;
	393222, 393223:
		//here you can add some special code for the three parameters
		pValue := pParameter^.dwValue;
		SysMemCpy((pValue + dwBitOffset/8), pData, MIN(DWORD_TO_BYTE(dwBitSize/8), UINT_TO_BYTE(pParameter^.wLen / 8)));			
		RETURN;
	327937: 
		(*
				Example for extended Diagnostic Acknowledge:
				- Parameter needs channel type "diagack": when user presses ACKNOWLEDGE WriteParameter is called
				- here only the flag is reset, so the diag message is not shown in the Editor any more  
		*)
        _connectorFlagController.DiagnosticAvailable := FALSE;
	//	IoMgrConfigResetDiagnosis(pConnector, Connectorflags.CF_CONNECTOR_DIAGNOSTIC_AVAILABLE);
		RETURN;
	ELSE
		pValue := pParameter^.dwValue; 
		SysMemCpy(pDest := pValue + dwBitOffset/8, pSrc := pData, pParameter^.wLen / 8);
END_CASE

IoDrvWriteParameter := Errors.ERR_FAILED;
END_METHOD

{attribute 'conditionalshow' := 'IoDrvDebug'}
METHOD IoDrvReadParameter : UDINT
VAR_INPUT
	pConnector : POINTER TO IoConfigConnector;
	pParameter : POINTER TO IoConfigParameter;
	pData : POINTER TO BYTE;
	dwBitSize : DWORD;
	dwBitOffset : DWORD;
END_VAR
VAR
	pValue : POINTER TO BYTE;
    pString : POINTER TO STRING;
    Result : UDINT := 0;
END_VAR
IF 	pConnector = 0 OR pParameter = 0 OR pData = 0 THEN
	IoDrvReadParameter := Errors.ERR_PARAMETER;
	RETURN;	
END_IF

IoDrvReadParameter := Errors.ERR_OK;

pValue := pParameter^.dwValue;
IF pValue <> 0 THEN
	CASE pParameter^.dwParameterId OF
		327936: 
			(*
				Example for extended Diagnostic:
				- Parameter needs channel type "diag": as long as connectorflag "CF_CONNECTOR_DIAGNOSTIC_AVAILABLE" is set, the IoDrvReadParameter will be called with the Parameter of channeltype "diag"
				- One may return a string that is shown in "status" editor in CODESYS			
			*)
         pString := IoMgrConfigGetParameterValuePointer(pParameter, ADR(Result));
         pString^ := 'Changeable ...';
	END_CASE
END_IF
// All standard parameters of our device are handled by the IO-manager!
IoDrvReadParameter := Errors.ERR_FAILED;
END_METHOD

{attribute 'conditionalshow' := 'IoDrvDebug'}
METHOD QueryInterface : POINTER TO POINTER TO BYTE
VAR_INPUT
	iid : DWORD; (* InterfaceID *)
	pResult : POINTER TO UDINT;	
END_VAR
VAR
END_VAR
QueryInterface_Count := QueryInterface_Count + 1;
IF iid = ITFID_ICmpIoDrv THEN
	QueryInterface := ADR(_IIoDrv);
	AddRef();
	IF (pResult <> 0) THEN
		pResult^ := Errors.ERR_OK;
	END_IF
	RETURN;	
ELSIF iid = ITFID_ICmpIoDrvParameter THEN
	QueryInterface := ADR(_IIoDrvParameter);
	AddRef();
	IF (pResult <> 0) THEN
		pResult^ := Errors.ERR_OK;
	END_IF	
	RETURN;	
ELSE
	QueryInterface := SUPER^.QueryInterface(iid, pResult);
END_IF
END_METHOD

{attribute 'conditionalshow' := 'IoDrvDebug'}
METHOD FB_Reinit : BOOL
VAR_INPUT
END_VAR
VAR
END_VAR
FB_Reinit_Count := FB_Reinit_Count + 1;
FB_Reinit := TRUE;
END_METHOD

{attribute 'conditionalshow' := 'IoDrvDebug'}
METHOD Initialize : UDINT
VAR_INPUT
	wModuleType : UINT;
	dwInstance : UDINT;
	pConnector : POINTER TO IoConfigConnector; 
END_VAR
VAR
END_VAR
Initialize_Count := Initialize_Count + 1;

m_wModuleType := wModuleType;
m_dwInstance := dwInstance;
m_Info.wModuleType := wModuleType;

Initialize := Errors.ERR_OK;
END_METHOD

{attribute 'conditionalshow' := 'IoDrvDebug'}
METHOD FB_Exit : BOOL
VAR_INPUT
	bInCopyCode: BOOL;	
END_VAR
VAR
END_VAR
FB_Exit_Count := FB_Exit_Count + 1;
FB_Exit := TRUE;
END_METHOD

{attribute 'conditionalshow' := 'IoDrvDebug'}
METHOD FB_Init : BOOL
VAR_INPUT
	bInitRetains: BOOL;
	bInCopyCode: BOOL;
END_VAR
VAR
	Result : UDINT;
END_VAR
FB_Init_Count := FB_Init_Count + 1;

m_Info.szDriverName := 'IoDrvMasterTemplateIEC';
m_Info.szVendorName := 'MyCompany';
m_Info.szDeviceName := 'MyCard';
m_Info.wModuleType := 40101;

_IIoDrv := THIS^;
_IIoDrvParameter := THIS^;

m_IBaseItf := THIS^;
m_hInterface := IoMgrRegisterInstance2(CLASSID_CCmpIoDrvTemplate, m_IBaseItf, ADR(Result));
FB_Init := TRUE;
END_METHOD

{attribute 'conditionalshow' := 'IoDrvDebug'}
METHOD IoDrvGetConnector : POINTER TO IoConfigConnector
VAR_INPUT
	pResult : POINTER TO RTS_IEC_RESULT;
END_VAR
VAR
END_VAR
IF m_pConnector = 0 THEN
	IF pResult <> 0 THEN
		pResult^ := Errors.ERR_FAILED;
	END_IF
	IoDrvGetConnector := 0;	
	RETURN;
END_IF
IF pResult <> 0 THEN
	pResult^ := Errors.ERR_OK;
END_IF
IoDrvGetConnector := m_pConnector;
END_METHOD

{attribute 'conditionalshow' := 'IoDrvDebug'}
METHOD Cleanup
VAR_INPUT
END_VAR
VAR

END_VAR
FreeScanData();
END_METHOD

{attribute 'conditionalshow' := 'IoDrvDebug'}
METHOD FreeScanData
VAR_INPUT
END_VAR
VAR
	pCurConnector : POINTER TO IoConfigConnector;
	pParameter : POINTER TO IoConfigParameter;	
	i : INT;
	j : INT;
END_VAR
//Free device scan data
IF _iScannedSlaves > 0 AND _pScanList <> 0 THEN
	pCurConnector := _pScanList;
	FOR i := 0 TO _iScannedSlaves - 1 DO
		pParameter := pCurConnector^.pParameterList;
		IF pParameter <> 0 THEN
			FOR j := 0 TO DWORD_TO_INT(pCurConnector^.dwNumOfParameters) - 1 DO
				IF (pParameter^.dwFlags AND IoStandard.ParameterValueFlags.PVF_POINTER) = IoStandard.ParameterValueFlags.PVF_POINTER THEN
					// dwValue is pointer
					IF pParameter^.dwValue <> 0 THEN
						SysMemFreeData(g_stComponentName, pParameter^.dwValue);
					END_IF
				END_IF
				pParameter := pParameter + SIZEOF(IoConfigParameter);	
			END_FOR
			SysMemFreeData(g_stComponentName, pCurConnector^.pParameterList);
		END_IF
		pCurConnector := pCurConnector + SIZEOF(IoStandard.IoConfigConnector);
	END_FOR
	SysMemFreeData(g_stComponentName, _pScanList);
	_pScanList := 0;
 	_iScannedSlaves := 0;
END_IF
END_METHOD

END_FUNCTION_BLOCK

// IoDrvMasterTemplateIEC/Function Blocks/IoDrvTemplateSlave
FUNCTION_BLOCK IoDrvTemplateSlave

VAR_INPUT
END_VAR

VAR_OUTPUT
END_VAR

VAR
	_bDeactivated : BOOL := TRUE;

    // There are 3 different slave types (differ in value of ParameterId="2"). T1 can have max 4 modules. T2 autoinserts 2 modules an just can have 2 modules. T3 has no modules an defines own in- and outputs. 
	_slaveType: DWORD := 0;
    // Value of ParameterId="256". Unique ID for the slave under the master. User hast to take care of this uniqueness. This number is needed to communicate with the counterpart (just a UDP messanger). 
	_slaveId: BYTE := 255;

    // Used to save the modules with their moduleID in a list. To access the correct module in the method IoDrvStartBusCylce fast. 
	_fal_shortcut2Modules :FixedArrayList; 
	
	// Type T3 variables, needed for the slave, which has no modules and fixed IO´s
    // (we could also use _fal_shortcut2Modules, which is unused in this case, but for the nameing ...
	_fal_ioParas :FixedArrayList; 
	
	// remember the connector and count, to set pConnector^.hIoDrv := 0 in UpdateConfigurationDestroy, because connector is not passed to it. 
	_pConnector: POINTER TO IoConfigConnector;	
	_nCount: DINT;
	
	_connectorFlagController : IoDrvUtility.ConnectorFlagController;
END_VAR

{attribute 'conditionalshow' := 'IoDrvDebug'}
METHOD Initialize : UDINT
VAR_INPUT
	wModuleType : UINT;
	dwInstance : UDINT;
	pConnector : POINTER TO IoConfigConnector; 
END_VAR
VAR
	{attribute 'no_init'}
	pParameter : POINTER TO IoConfigParameter;
	{attribute 'no_init'}
	p_dwParValue : POINTER TO XWORD;
	Result : UDINT := 0;
	
END_VAR
(* Enter the thispointer to an implicit parameter in the configuration data. *)
pParameter := ConfigGetParameter(pConnector, 1);
IF pParameter <> 0 THEN
	p_dwParValue := ConfigGetParameterValuePointer(pParameter,ADR(Result));
	IF p_dwParValue <> 0 THEN
		p_dwParValue^ := THIS;
	END_IF
END_IF
END_METHOD

METHOD UpdateConfigurationCreate : UDINT
VAR_INPUT
	pConnector : POINTER TO IoConfigConnector; 
	hInterface : RTS_IEC_HANDLE;	
	nCount : DINT;
END_VAR
VAR_OUTPUT
	xDisabled : BOOL;
END_VAR
VAR
	p_dwParValueModule : POINTER TO IoDrvTemplateModule;
	pDummy			: POINTER TO XWORD;
	pParameter : POINTER TO IoConfigParameter;

	i: DWORD := 0;
	
	nCountRemember : DINT;
	pChild : POINTER TO IoConfigConnector;		
	Result : UDINT := 0;

	searchParam: UDINT;
	moduleCounter : UDINT := 0;
	myIecResult : RTS_IEC_Result;
	moduleIter : POINTER TO Module;
	
	pIoEntry : POINTER TO IoEntry;
	xModuleDisabled : BOOL;
END_VAR
UpdateConfigurationCreate := Errors.ERR_OK;
// just getting called, when Connector is enabled
_bDeactivated := FALSE;
_pConnector := pConnector;
_nCount := nCount;
pConnector^.hIoDrv := hInterface;	// Registered instance handle of the IO-driver, that operates this device respectively this connector

_connectorFlagController.Init(pConnector := _pConnector, uiNCount := _nCount, xSetChildren := TRUE);
_connectorFlagController.DiagProvider := TRUE;
_connectorFlagController.AutoSetErrorClearedFlag := TRUE;
IF _connectorFlagController.State = IoDrvUtility.ConnectorState.DISABLED THEN
	xDisabled := TRUE;
	RETURN;
END_IF

pParameter := IoMgrConfigGetParameter(pConnector, 256); // get Slave-ID
IF pParameter <> 0 THEN
	_slaveId := IoMgrConfigGetParameterValueByte(pParameter, ADR(Result));
ELSE
	UpdateConfigurationCreate := Errors.ERR_FAILED; // missing Slave-ID
	RETURN;
END_IF

pParameter := IoMgrConfigGetParameter(pConnector, 2);
IF pParameter <> 0 THEN
	_slaveType := IoMgrConfigGetParameterValueDword(pParameter, ADR(myIecResult));
	CASE _slaveType OF // Slave Type over default values in xml DeviceDescription
		1, 2: // variable, variable autoinsert
			// can have more childs (modules)
			moduleCounter := 0;		
			
			pConnector := IoMgrConfigGetFirstChild(pConnector, ADR(nCount), pConnector); // getChild x2 is the next entry in device tree -> a device with subnodes has 2 connectors in xml! special case for this is, when you have a module, wich could be used with different slaves, which have different connectors ...
			pConnector^.hIoDrv := hInterface;
            nCountRemember := nCount; // saving the position to runt through the modules again to fill the reserved space
						
			pChild := IoMgrConfigGetFirstChild(pConnector, ADR(nCount), pConnector);
			WHILE (pChild <> 0) DO
				// children of slaves are IoDrvTemplateModule FB´s -> call them UpdateConfigurationCreate(...)
				pParameter := IoMgrConfigGetParameter(pChild, 1); 
				IF pParameter <> 0 THEN			
					pDummy := ConfigGetParameterValuePointer(pParameter,ADR(Result));
					p_dwParValueModule :=  pDummy^;
					IF p_dwParValueModule <> 0 THEN
						UpdateConfigurationCreate := UpdateConfigurationCreate OR p_dwParValueModule^.UpdateConfigurationCreate(pConnector := pChild, hInterface, nCount, xDisabled => xModuleDisabled);
						IF NOT xModuleDisabled THEN
							moduleCounter := moduleCounter + 1;
						END_IF
					END_IF
				END_IF

				pChild := IoMgrConfigGetNextChild(pChild, ADR(nCount), pConnector);
			END_WHILE
			
			//any modules with Create problems? then stop
			IF (UpdateConfigurationCreate <> Errors.ERR_OK) THEN
				RETURN;
			END_IF
			
			// reserve space to save module 
			IF( NOT _fal_shortcut2Modules.Create(moduleCounter, SIZEOF(Module), g_stComponentName) ) THEN 
				UpdateConfigurationCreate := Errors.ERR_NOMEMORY; // no space ....
				RETURN;
			END_IF

			// fill the space with the values
			i := 0;
			nCount := nCountRemember;
			pChild := IoMgrConfigGetFirstChild(pConnector, ADR(nCount), pConnector);
			WHILE (pChild <> 0) DO
				// childs of slaves are IoDrvTemplateModule FB´s -> call them UpdateConfigurationCreate(...)
				pParameter := IoMgrConfigGetParameter(pChild, 1); 
				IF pParameter <> 0 THEN			
					pDummy := ConfigGetParameterValuePointer(pParameter,ADR(Result));
					p_dwParValueModule :=  pDummy^;
					IF p_dwParValueModule <> 0 THEN
						IF NOT p_dwParValueModule^.IsDisabled THEN
							moduleIter := _fal_shortcut2Modules.Get(i);
							i := i + 1;
							moduleIter^.moduleInstance := p_dwParValueModule;
						END_IF
					END_IF
				END_IF
				pChild := IoMgrConfigGetNextChild(pChild, ADR(nCount), pConnector);
			END_WHILE
			
		3: // no module
		// IO´s are in the slave -> no children (modules)
			(*
			Here we have a slave with input and output channels. Now the parameters for this slave could be on fixed ID´s and have a fixed size (Parameter 2000 is an input and a byte).
			If this is going to change to 2 inputs with the size of a WORD, then the XML file changes and the code, which would be below this comment, would also need to be changed. 
			But we can act dynamically, like its done here. We define, that inputs-parametersIds are between 2000-2999 and outputs-parametersIds between 3000-3999. Over wLen we can 
			check the size of the parameter to allocate space for the doublebuffer:
			Now we need some space to doublebuffer the values (pParameter^.dwValue). To save the adress of the doublebuffer, we have pParameter^.dwDriverSpecific, which is a XDWORD.
			E.g. if we have a byte of Inputvalues, we need a place to safe this values, when we receive them on the bus. This copies are getting copied to the actual values, when 
			the ReadInputs process begins. The same is valid for outputs. If we have 1 byte output and the WriteOutputs process begins, we need a place to save the values, because 
			we "can´t" send them directy over the bussystem (i.e. CAN -> somebody else is sending whith lower ID). 
			At this point we have time to allocate space i.e. over sysmem, because we are not at a time-critical point (don´t forget to free: When IoDrvUpdateConfiguration -> if( pConnectorList = 0) ).
			The download is finished and now we are getting called. We could also use static memory over an array i.e. BYTE[Max Slaves*IOsize]. Or we can also use the pParameter^.dwDriverSpecific to
			save our values directly in there, what is done in this example. This is possible, because we can assure that the IO data are smaller or equal to 16 Bit (<=sizeof(XWORD)). 
			Another possibility is, to define another identical parameter, which is not visible to the user, to doublebuffer the value in there.  
			*)
			
			// has some fixed (at runtime) in- or/and outputs, can be added in the xml file (consecutive number)
			// ParameterId="2000" - 2999 are digital inputs
			// ParameterId="3000" - 3999 are digital outputs
			
			// count inputs & outputs, to know how much memory we need to save shortcuts
			i :=0;
			searchParam := PARAMS_IODRVTEMPLATEMASTER.START_OF_INPUTPARAMS; // inputcount
			REPEAT
				pParameter := IoMgrConfigGetParameter(pConnector, searchParam);
				IF pParameter <> CAA.gc_pNull THEN
					i := i + 1;
					searchParam := searchParam + 1;
				END_IF
			UNTIL 
				(pParameter = CAA.gc_pNull) OR (searchParam >= PARAMS_IODRVTEMPLATEMASTER.END_OF_INPUTPARAMS)
			END_REPEAT;
			searchParam := PARAMS_IODRVTEMPLATEMASTER.START_OF_OUTPUTPARAMS; // outputcount
			REPEAT
				pParameter := IoMgrConfigGetParameter(pConnector, searchParam);
				IF pParameter <> CAA.gc_pNull THEN
					i := i + 1;
					searchParam := searchParam + 1;
				END_IF
			UNTIL 
				(pParameter = CAA.gc_pNull) OR (searchParam >= PARAMS_IODRVTEMPLATEMASTER.END_OF_OUTPUTPARAMS)
			END_REPEAT;
			
			// get space to create shortcuts
			IF( NOT _fal_ioParas.Create(i, SIZEOF(IoEntry), g_stComponentName) ) THEN
				UpdateConfigurationCreate := Errors.ERR_NOMEMORY; // no space ....
				RETURN;
			END_IF
				
			// fill with shortcuts
			i :=0; 
			searchParam := PARAMS_IODRVTEMPLATEMASTER.START_OF_INPUTPARAMS; // input fill
			REPEAT
				pParameter := IoMgrConfigGetParameter(pConnector, searchParam);
				IF pParameter <> CAA.gc_pNull THEN
					pIoEntry := _fal_ioParas.Get(i);
					pIoEntry^.pParameter := pParameter;
					pIoEntry^.ioType := IoType.INPUT;
					i := i + 1;
					searchParam := searchParam + 1;
				END_IF
			UNTIL 
				(pParameter = CAA.gc_pNull) OR (searchParam >= PARAMS_IODRVTEMPLATEMASTER.END_OF_INPUTPARAMS)
			END_REPEAT;
			searchParam := PARAMS_IODRVTEMPLATEMASTER.START_OF_OUTPUTPARAMS; // output fill
			REPEAT
				pParameter := IoMgrConfigGetParameter(pConnector, searchParam);
				IF pParameter <> CAA.gc_pNull THEN
					pIoEntry := _fal_ioParas.Get(i);
					pIoEntry^.pParameter := pParameter;
					pIoEntry^.ioType := IoType.OUTPUT;
					i := i + 1;
					searchParam := searchParam + 1;
				END_IF
			UNTIL 
				(pParameter = CAA.gc_pNull) OR (searchParam >= PARAMS_IODRVTEMPLATEMASTER.END_OF_OUTPUTPARAMS)
			END_REPEAT;
			
			// now we need to doublebuffer the parameters, e.g. if an input is recived over the bussystem, we dont wont do directy write it into the value. This should be done in IoDrvReadInputs. Same for outputs.
			// To reach doublebuffering, we need th same space as the value has (wLen) for each IO ...
			IF _fal_ioParas.Size > 0 THEN
				FOR i:=0 TO _fal_ioParas.Size - 1 DO
					pIoEntry := _fal_ioParas.Get(i);
					IF( pIoEntry^.pParameter^.wLen MOD 8) <> 0 THEN // wLen is in Bits, getting from heap is in bytes
						pIoEntry^.pParameter^.dwDriverSpecific := SysMemAllocData(g_stComponentName, (pIoEntry^.pParameter^.wLen / 8) +1 , ADR(myIecResult));  // dont forget to delete -> UpdateConfigurationDestroy
					ELSE
						pIoEntry^.pParameter^.dwDriverSpecific := SysMemAllocData(g_stComponentName, (pIoEntry^.pParameter^.wLen / 8)    , ADR(myIecResult)); 
					END_IF
					IF (myIecResult <> Errors.ERR_OK) THEN
						UpdateConfigurationCreate := Errors.ERR_NOMEMORY; // no space
						RETURN;
					END_IF
				END_FOR
			END_IF	
	END_CASE
	
	_connectorFlagController.State := IoDrvUtility.ConnectorState.RUNNING;
ELSE
	UpdateConfigurationCreate := Errors.ERR_FAILED; // missing Type
	RETURN;
END_IF
END_METHOD

METHOD UpdateConfigurationDestroy
VAR_INPUT
END_VAR
VAR
	moduleIter: POINTER TO Module;	
	i: DWORD := 0;
	pIoEntry : POINTER TO IoEntry;
	pConnector: POINTER TO IoConfigConnector;
END_VAR
_pConnector^.hIoDrv := 0;

CASE _slaveType OF // Slave Type over default values in xml DeviceDescription
	1, 2: // varbiable, variable autoinsert
		// unregister driver
		pConnector := IoMgrConfigGetFirstChild(_pConnector, ADR(_nCount), _pConnector); // getChild x2 is the next entry in device tree -> a device with subnodes has 2 connectors in xml! special case for this is, when you have a module, wich could be used with different slaves, which have different connectors ...
		pConnector^.hIoDrv := 0;
		//Go through all childs of the device
		IF _fal_shortcut2Modules.Size > 0 THEN
			FOR i:=0 TO _fal_shortcut2Modules.Size - 1 DO
				moduleIter := _fal_shortcut2Modules.Get(i);
				moduleIter^.moduleInstance^.UpdateConfigurationDestroy(); // childs of slaves are IoDrvTemplateModule FB´s -> call them UpdateConfigurationDestroy(...)
			END_FOR
		END_IF
		_fal_shortcut2Modules.Destroy();// delete shortcut list to slaves 	
	3: // no module
		IF _fal_ioParas.Size > 0 THEN
			FOR i:=0 TO _fal_ioParas.Size - 1 DO
				pIoEntry := _fal_ioParas.Get(i);
				SysMemFreeData(g_stComponentName, pIoEntry^.pParameter^.dwDriverSpecific);			
			END_FOR
		END_IF
		_fal_ioParas.Destroy();
	
END_CASE 

// reset var´s (needed when reconfigure is activated)
_bDeactivated := TRUE;
_slaveType := 0;
_slaveId := 255;
_pConnector := 0;	
_nCount := 0;
END_METHOD

METHOD StartBusCycle
VAR_INPUT
END_VAR

VAR_IN_OUT
	udpIO: UdpIO;
END_VAR

VAR
	i : DWORD;
	moduleIter : POINTER TO Module;
	pIoEntry1, pIoEntry2 : POINTER TO IoEntry;
END_VAR
CASE _slaveType OF // Slave Type over default values in xml DeviceDescription
	1, 2: // varbiable, variable autoinsert
		
		IF _fal_shortcut2Modules.Size > 0 THEN
			FOR i:=0 TO _fal_shortcut2Modules.Size - 1 DO
				moduleIter := _fal_shortcut2Modules.Get(i);
				IF(udpIO.r_BytesReceived > 1) THEN
					IF( moduleIter^.moduleInstance^.ModuleID = udpIO.r_udpInBuffer^.Get(1)^  ) THEN // modulId is the received one?
						udpIO.s_udpOutBuffer^.Get(0)^ := SlaveID; // put the slaveID in the first byte of the ouput buffer, if the module is sending this entry is needed
						moduleIter^.moduleInstance^.StartBusCycle(udpIO);
					END_IF
				END_IF
			END_FOR
		END_IF
			
	3: // no module
		
		// is not controlled over udp ... copy the inputs to the outputs	
	
		pIoEntry1 := _fal_ioParas.Get(0); // input --> preknown because i know that there should be 1 input and 1 ouput in the xml file and first are filled the inputs and then the ouputs ... so 0 is the input and 1 is the ouput
		pIoEntry2 := _fal_ioParas.Get(1); // ouput 
		
		SysMem.SysMemCpy(pIoEntry1^.pParameter^.dwDriverSpecific, pIoEntry2^.pParameter^.dwDriverSpecific, 1);

END_CASE
END_METHOD

PROPERTY SlaveID : BYTE
GET
SlaveID := _slaveId;
END_GET
END_PROPERTY

PROPERTY INTERNAL IsDisabled : BOOL
GET
IsDisabled := _connectorFlagController.State = IoDrvUtility.ConnectorState.DISABLED;
END_GET
END_PROPERTY

END_FUNCTION_BLOCK

// IoDrvMasterTemplateIEC/Function Blocks/IoDrvTemplateModule
FUNCTION_BLOCK IoDrvTemplateModule

VAR_INPUT
END_VAR

VAR_OUTPUT
END_VAR

VAR
	_bDeactivated : BOOL := TRUE;
    
    // Value of ParameterId="256". Unique ID for the module under the slave. User hast to take care of this uniqueness. This number is needed to communicate with the counterpart (just a UDP messanger). 
	_moduleID : BYTE;
    // Used to save the IO´s. To access them fast in the method IoDrvStartBusCylce. 
	_fal_ioParas :FixedArrayList;
	
	// remember the connector and count, to set pConnector^.hIoDrv := 0 in UpdateConfigurationDestroy, because connector is not passed to it. 
	_pConnector: POINTER TO IoConfigConnector;	
	_nCount: DINT;
	
	_connectorFlagController : IoDrvUtility.ConnectorFlagController;
	
END_VAR

{attribute 'conditionalshow' := 'IoDrvDebug'}
METHOD Initialize : UDINT
VAR_INPUT
	wModuleType : UINT;
	dwInstance : UDINT;
	pConnector : POINTER TO IoConfigConnector; 
END_VAR
VAR
	{attribute 'no_init'}
	pParameter : POINTER TO IoConfigParameter;
	{attribute 'no_init'}
	p_dwParValue : POINTER TO XWORD;
	Result : UDINT := 0;
	
END_VAR
(* Enter the thispointer to an implicit parameter in the configuration data. *)
pParameter := ConfigGetParameter(pConnector, 1);
IF pParameter <> 0 THEN
	p_dwParValue := ConfigGetParameterValuePointer(pParameter,ADR(Result)); 
	IF p_dwParValue <> 0 THEN
		p_dwParValue^ := THIS; // writing in dwDriverSpecific (XWORD)
	END_IF
END_IF
END_METHOD

METHOD UpdateConfigurationCreate: UDINT
VAR_INPUT
	pConnector : POINTER TO IoConfigConnector; 
	hInterface : RTS_IEC_HANDLE;	
	nCount : DINT;
END_VAR
VAR_OUTPUT
	xDisabled : BOOL;
END_VAR
VAR
	pParameter : POINTER TO IoConfigParameter;
	pChild : POINTER TO IoConfigConnector;		
	i: DWORD := 0;
	counter : UDINT := 0;
	searchParam: UDINT;
	myIecResult : RTS_IEC_Result;
	pIoEntry : POINTER TO IoEntry;
END_VAR
UpdateConfigurationCreate := Errors.ERR_OK;
// pConnector is _pConnector
			
// just getting called, when Connector is enabled
_bDeactivated := FALSE;
_pConnector := pConnector;	
_nCount := nCount;
	
pConnector^.hIoDrv := hInterface;	// Registered instance handle of the IO-driver, that operates this device respectively this connector

_connectorFlagController.Init(pConnector := _pConnector, uiNCount := _nCount, xSetChildren := FALSE);
_connectorFlagController.DiagProvider := TRUE;
_connectorFlagController.AutoSetErrorClearedFlag := TRUE;

IF _connectorFlagController.State = IoDrvUtility.ConnectorState.DISABLED THEN
	xDisabled := TRUE;
	RETURN;
END_IF

pParameter := IoMgrConfigGetParameter(pConnector, 256); // get Module-ID
IF pParameter <> 0 THEN
	_moduleID := IoMgrConfigGetParameterValueByte(pParameter, ADR(myIecResult));
ELSE
	UpdateConfigurationCreate := Errors.ERR_FAILED; // missing Module-ID
	RETURN;
END_IF			

// now here is the same valid as in IoDrvTemplateSlave(FB)->Init (Folder)-> UpdateConfigurationCreate (Method)-> Type 3 of slave (search for: "3: // no module")
// for the example we use the same addressing scheme (ip/moduleId/parameterID - ip/moduleId/slaveID/parameterID) for the module as for the slave type 3.

// has some fixed (at runtime) in- or/and outputs, can be added in the xml file (consecutive number)
			// ParameterId="2000" - 2999 are digital inputs
			// ParameterId="3000" - 3999 are digital outputs
			
			// count inputs & outputs, to know how much memory we need to save shortcuts
counter :=0;
searchParam := PARAMS_IODRVTEMPLATEMASTER.START_OF_INPUTPARAMS; // inputcount
REPEAT
	pParameter := IoMgrConfigGetParameter(pConnector, searchParam);
	IF pParameter <> CAA.gc_pNull THEN
		counter := counter + 1;
		searchParam := searchParam + 1;
	END_IF
UNTIL 
	(pParameter = CAA.gc_pNull) OR (searchParam >= PARAMS_IODRVTEMPLATEMASTER.END_OF_INPUTPARAMS)
END_REPEAT;
searchParam := PARAMS_IODRVTEMPLATEMASTER.START_OF_OUTPUTPARAMS; // outputcount
REPEAT
	pParameter := IoMgrConfigGetParameter(pConnector, searchParam);
	IF pParameter <> CAA.gc_pNull THEN
		counter := counter + 1;
		searchParam := searchParam + 1;
	END_IF
UNTIL 
	(pParameter = CAA.gc_pNull) OR (searchParam >= PARAMS_IODRVTEMPLATEMASTER.END_OF_OUTPUTPARAMS)
END_REPEAT;
	
// get space to create shortcuts
IF( NOT _fal_ioParas.Create(counter, SIZEOF(IoEntry), g_stComponentName) ) THEN
	UpdateConfigurationCreate := Errors.ERR_NOMEMORY; // no space ....
	RETURN;
END_IF
	
// fill with shortcuts
i :=0; 
searchParam := PARAMS_IODRVTEMPLATEMASTER.START_OF_INPUTPARAMS; // input fill
REPEAT
	pParameter := IoMgrConfigGetParameter(pConnector, searchParam);
	IF pParameter <> CAA.gc_pNull THEN
		pIoEntry := _fal_ioParas.Get(i);
		pIoEntry^.pParameter := pParameter;
		pIoEntry^.ioType := IoType.INPUT;
		i := i + 1;
		searchParam := searchParam + 1;
	END_IF
UNTIL 
	(pParameter = CAA.gc_pNull) OR (searchParam >= PARAMS_IODRVTEMPLATEMASTER.END_OF_INPUTPARAMS)
END_REPEAT;
searchParam := PARAMS_IODRVTEMPLATEMASTER.START_OF_OUTPUTPARAMS; // output fill
REPEAT
	pParameter := IoMgrConfigGetParameter(pConnector, searchParam);
	IF pParameter <> CAA.gc_pNull THEN
		pIoEntry := _fal_ioParas.Get(i);
		pIoEntry^.pParameter := pParameter;
		pIoEntry^.ioType := IoType.OUTPUT;
		i := i + 1;
		searchParam := searchParam + 1;
	END_IF
UNTIL 
	(pParameter = CAA.gc_pNull) OR (searchParam >= PARAMS_IODRVTEMPLATEMASTER.END_OF_OUTPUTPARAMS)
END_REPEAT;
			
// now we need to doublebuffer the parameters, e.g. if an input is recived over the bussystem, we dont wont do directy write it into the value. This should be done in IoDrvReadInputs. Same for outputs.
// To reach doublebuffering, we need th same space as the value has (wLen) for each IO ...
IF _fal_ioParas.Size > 0 THEN
	FOR i:=0 TO _fal_ioParas.Size - 1 DO
		pIoEntry := _fal_ioParas.Get(i);
		IF( pIoEntry^.pParameter^.wLen MOD 8) <> 0 THEN // wLen is in Bits, getting from heap is in bytes
			pIoEntry^.pParameter^.dwDriverSpecific := SysMemAllocData(g_stComponentName, (pIoEntry^.pParameter^.wLen / 8) +1 , ADR(myIecResult));  // dont forget to delete -> UpdateConfigurationDestroy
			ELSE
				pIoEntry^.pParameter^.dwDriverSpecific := SysMemAllocData(g_stComponentName, (pIoEntry^.pParameter^.wLen / 8)    , ADR(myIecResult)); 
			END_IF
			IF (myIecResult <> Errors.ERR_OK) THEN
			UpdateConfigurationCreate := Errors.ERR_NOMEMORY; // no space
			RETURN;
		END_IF
	END_FOR
END_IF

_connectorFlagController.State := IoDrvUtility.ConnectorState.RUNNING;
END_METHOD

METHOD UpdateConfigurationDestroy
VAR_INPUT
END_VAR
VAR
	i: DWORD := 0;
	pIoEntry : POINTER TO IoEntry;
END_VAR
_pConnector^.hIoDrv := 0;

IF _fal_ioParas.Size > 0 THEN
	FOR i:=0 TO _fal_ioParas.Size - 1 DO
		pIoEntry := _fal_ioParas.Get(i);
		SysMemFreeData(g_stComponentName, pIoEntry^.pParameter^.dwDriverSpecific);			
	END_FOR
END_IF

_fal_ioParas.Destroy();

_bDeactivated := TRUE;
_moduleID := 0;
_pConnector := 0;	
_nCount := 0;
END_METHOD

METHOD StartBusCycle
VAR_INPUT
END_VAR

VAR_IN_OUT
	udpIO: UdpIO;
END_VAR

VAR
	i, j, paraId: DWORD := 0;
	pIoEntry : POINTER TO IoEntry;
	
	pHelper: POINTER TO  BYTE;
	
END_VAR
IF(udpIO.r_BytesReceived > 5) THEN // enough bytes received?
	paraId := SHL( BYTE_TO_DWORD(udpIO.r_udpInBuffer^.Get(5)^), 24) OR SHL( BYTE_TO_DWORD(udpIO.r_udpInBuffer^.Get(4)^), 16) OR  SHL( BYTE_TO_DWORD(udpIO.r_udpInBuffer^.Get(3)^), 8) OR BYTE_TO_DWORD(udpIO.r_udpInBuffer^.Get(2)^); // get the ParameterId out of the received udp payload
	IF _fal_ioParas.Size > 0 THEN
		FOR i:=0 TO _fal_ioParas.Size - 1 DO // search the given parameter
			pIoEntry := _fal_ioParas.Get(i);
			IF(paraId = pIoEntry^.pParameter^.dwParameterId) THEN // parameterId found
				pHelper := pIoEntry^.pParameter^.dwDriverSpecific; // get pointer to the data (the doublebuffer -> valuepointer is written or read in IoDrvWriteOutputs or IoDrvReadInputs. 
				CASE pIoEntry^.ioType OF
					IoType.INPUT: // if input, then write the new input values
						IF(udpIO.r_BytesReceived > (5 + pIoEntry^.pParameter^.wLen / 8)) THEN // enough bytes received to fill the value?
							FOR j:=1 TO  pIoEntry^.pParameter^.wLen / 8 DO
								pHelper^ := udpIO.r_udpInBuffer^.Get(j + 5)^;
								pHelper := pHelper + 1;
							END_FOR
						END_IF
					IoType.OUTPUT: // if ouput, then send back the output value
						// first byte was added by slave already (slaveId (8Bit))
						udpIO.s_udpOutBuffer^.Get(1)^ := ModuleID; // (moduleId (8Bit))
						udpIO.s_udpOutBuffer^.Get(2)^ := DWORD_TO_BYTE( pIoEntry^.pParameter^.dwParameterId) ; // parameterId (32Bit)
						udpIO.s_udpOutBuffer^.Get(3)^ := DWORD_TO_BYTE( SHR(pIoEntry^.pParameter^.dwParameterId, 8));
						udpIO.s_udpOutBuffer^.Get(4)^ := DWORD_TO_BYTE( SHR(pIoEntry^.pParameter^.dwParameterId, 16));
						udpIO.s_udpOutBuffer^.Get(5)^ := DWORD_TO_BYTE( SHR(pIoEntry^.pParameter^.dwParameterId, 24));
						FOR j:=1 TO  pIoEntry^.pParameter^.wLen / 8 DO
							udpIO.s_udpOutBuffer^.Get(5 +j)^ := pHelper^;
							pHelper := pHelper + 1;
						END_FOR
						IF( pIoEntry^.pParameter^.wLen MOD 8 <> 0) THEN
							udpIO.s_udpOutBuffer^.Get(5 +j)^ := pHelper^; // add one more byte for the last bits ....
							// 1 byte longer than normal ....
							udpIO.s_udpSender^(xExecute := TRUE, udiTimeOut := 0, hPeer := udpIO.s_udpPeer^.hPeer, ipAddr := udpIO.s_ipSendTo^, uiPort := udpIO.s_portSendTo, szSize :=  pIoEntry^.pParameter^.wLen / 8 + 7, pData := udpIO.s_udpOutBuffer^.Get(0) );
						ELSE
							// normal
							udpIO.s_udpSender^(xExecute := TRUE, udiTimeOut := 0, hPeer := udpIO.s_udpPeer^.hPeer, ipAddr := udpIO.s_ipSendTo^, uiPort := udpIO.s_portSendTo, szSize :=  pIoEntry^.pParameter^.wLen / 8 + 6, pData := udpIO.s_udpOutBuffer^.Get(0) );
						END_IF
						IF(udpIO.s_udpSender^.xDone OR udpIO.s_udpSender^.xError) THEN // sending only on rising edge
							udpIO.s_udpSender^(xExecute := FALSE);
						END_IF
				END_CASE
			END_IF
		END_FOR
	END_IF
END_IF
END_METHOD

PROPERTY ModuleID : BYTE
GET
ModuleID := _moduleID;
END_GET
END_PROPERTY

PROPERTY INTERNAL IsDisabled : BOOL
GET
IsDisabled := _connectorFlagController.State = IoDrvUtility.ConnectorState.DISABLED;
END_GET
END_PROPERTY

END_FUNCTION_BLOCK

// IoDrvMasterTemplateIEC/Function Blocks/IoDrvTemplateMasterDiag
//This function block implements the diagnosis code for CAA Device Diagnosis.
{attribute 'no_assign'}
{attribute 'conditionalshow_all_locals' := 'IoDrvDebug'}
FUNCTION_BLOCK IoDrvTemplateMasterDiag EXTENDS IoDrvTemplateMaster IMPLEMENTS DED.IDevice2, DED.IBus, DED.IStack, DED.IReconfigureProvider
VAR_INPUT
END_VAR
VAR_OUTPUT
END_VAR
VAR
	_diag : DED.CAADiagnosisBase;
	_tree : DED.CAADiagTreeBase;
	_reconfig : DED.CAAReconfigureBase; //optional
END_VAR

(*Returns the number of childs below the current node*)
PROPERTY ChildNodeCount : CAA.COUNT
GET
ChildNodeCount := _tree.ChildNodeCount;
END_GET
END_PROPERTY

PROPERTY Connector : POINTER TO IoStandard.IoConfigConnector
GET
Connector := _tree.Connector;
END_GET
END_PROPERTY

(*This property returns if the node is enabled in the device tree. The setter can be used to change the Enabled flag. If enabling/disabling is not supported on the node the flag’s value will not change.*)
PROPERTY Enable : BOOL
GET
Enable := _tree.Enable;
END_GET
SET
_tree.Enable := Enable;
END_SET
END_PROPERTY

(*Returns the first child node below the current one*)
PROPERTY FirstChildNode : DED.INode
GET
FirstChildNode := _tree.FirstChildNode;
END_GET
END_PROPERTY

PROPERTY Index : UDINT
GET
Index := _tree.Index;
END_GET
SET
_tree.Index := Index;
END_SET
END_PROPERTY

(* returns true, if the current node is the root (plc) node, otherwise false*)
PROPERTY IsRootNode : BOOL
GET
IsRootNode := _tree.IsRootNode;
END_GET
END_PROPERTY

(* returns the next sibling node at the same level
 used for step through all nodes*)
PROPERTY NextSiblingNode : DED.INode
GET
NextSiblingNode := _tree.NextSiblingNode;
END_GET
END_PROPERTY

(* Returns the parent node or zero if already the root node is reached*)
PROPERTY ParentNode : DED.INode
GET
ParentNode := _tree.ParentNode;
END_GET
END_PROPERTY

(* Returns the number of sibling (same level) nodes*)
PROPERTY SiblingNodeCount : CAA.COUNT
GET
SiblingNodeCount := _tree.SiblingNodeCount;
END_GET
END_PROPERTY

{attribute 'hide'}
METHOD GetChild : DED.INode
VAR_INPUT
	udiIndex	: UDINT;
END_VAR
GetChild:= _tree.GetChild(udiIndex);
END_METHOD

{attribute 'hide'}
METHOD Initialize_Diag : UDINT
VAR_INPUT
	pConnector	: POINTER TO IoStandard.IoConfigConnector;
	nConnectorCount	: DINT;
	parent	: POINTER TO DED.INode;
	children	: POINTER TO DED.INode;
	udiChildCount	: UDINT;
END_VAR
//general initialization code: do not remove!
_tree.Initialize_Diag(pConnector, nConnectorCount, parent, children, udiChildCount);
_diag.Initialize_Diag(pConnector, nConnectorCount);

//if IReconfigureProvider is implemented
_reconfig.Initialize_Diag(THIS^);
END_METHOD

{attribute '''NORMAL__COMMENT' := 'Returns the fieldbus specific device state; interpretation is fieldbus dependent'}
(*Returns the fieldbus specific device state; interpretation is fieldbus dependent*)
METHOD GetSpecificDeviceState : DED.ERROR (* eError *)
VAR_INPUT
	(*Pointer to memory*)
	pData	: CAA.PVOID;
	(*Size of memory in bytes where pData is pointing to*)
	szSize	: CAA.SIZE;
END_VAR
VAR_OUTPUT
	(*Number of Bytes written to pData*)
	szCount	: CAA.SIZE;
END_VAR
GetSpecificDeviceState := DED.ERROR.NOT_SUPPORTED;
END_METHOD

(*Starts, stops or resets a device*)
METHOD SetCommunicationState : DED.ERROR (* eError *)
VAR_INPUT
	eRequestedState	: DED.DEVICE_TRANSITION_STATE;
END_VAR
IF CheckCurrentSupportedCommunicationState(eRequestedState) THEN
	CASE eRequestedState OF
		DED.DEVICE_TRANSITION_STATE.RESET:
			//TODO: Send a reset command to the device.
		DED.DEVICE_TRANSITION_STATE.START:
			//TODO: Send a start command to the device.
		DED.DEVICE_TRANSITION_STATE.STOP:
			//TODO: Send a stop command to the device.
	END_CASE
ELSE
	SetCommunicationState := DED.ERROR.OPERATION_INVALID;
END_IF
END_METHOD

(*Returns the device information of the current node*)
METHOD GetDeviceInfo : DED.ERROR (*eError*)
VAR_IN_OUT
	(*Device information struct*)
	deiInfo	: DED.DEVICE_INFO;
END_VAR
//base implementation supports all 3S specific fieldbusses.
GetDeviceInfo := _diag.GetDeviceInfo(deiInfo);
END_METHOD

{attribute 'hide'}
(* Returns the device error of the current node; you can also use functionblock GetDeviceError.*)
METHOD GetDeviceErrorAsync : DED.PROC_STATE (* eState *)
VAR_INPUT
	(*eCommand*)
	eCmd	: DED.PROC_CMD;
END_VAR
VAR_IN_OUT
	(*error struct*)
	eriDeviceError	: DED.ERROR_INFO;
END_VAR
VAR_OUTPUT
	(*error code if method fails*)
	eError	: DED.ERROR;
END_VAR
//optional method; base implementation returns NOT_SUPPORTED
GetDeviceErrorAsync := _diag.GetErrorAsync(eCmd, eriDeviceError, eError => eError);
END_METHOD

{attribute 'hide'}
(*Returns the specific device error of the current node; interpretation is fieldbus-dependent; you can also use functionblock GetSpecificDeviceError*)
METHOD GetSpecificDeviceErrorAsync : DED.PROC_STATE (* eState *)
VAR_INPUT
	(*eCommand*)
	eCmd	: DED.PROC_CMD;
	(*Pointer to memory*)
	pData	: CAA.PVOID;
	(*Size of memory in bytes where pData is pointing to*)
	szSize	: CAA.SIZE;
END_VAR
VAR_OUTPUT
	(*Number of Bytes written to pData*)
	szCount	: CAA.SIZE;
	(*error code if method fails*)
	eError	: DED.ERROR;
END_VAR
//optional method; base implementation returns NOT_SUPPORTED
GetSpecificDeviceErrorAsync := _diag.GetSpecificDeviceErrorAsync(eCmd,pData, szSize, szCount=>szCount, eError => eError);
END_METHOD

{attribute '''NORMAL__COMMENT' := 'Returns a DiagnosisInfo if xDiagnosisInfoAvailable of GetDeviceState was true.'}
(*Returns a DiagnosisInfo if xDiagnosisInfoAvailable of GetDeviceState was true.*)
METHOD GetDeviceDiagnosisInfo : DED.ERROR (*eError*)
VAR_INPUT
	(*Pointer to memory*)
	pData	: CAA.PVOID;
	(*Size of memory in bytes where pData is pointing to*)
	szSize	: CAA.SIZE;
END_VAR
VAR_OUTPUT
	(*Number of Bytes written to pData*)
	szCount	: CAA.SIZE;
END_VAR
//This is an optional method. Return device specific diagnostic information
GetDeviceDiagnosisInfo := DED.ERROR.NOT_SUPPORTED;
END_METHOD

(*Returns the state of the device; if device state is ERROR further information can be read by GetDeviceError*)
METHOD GetDeviceState : DED.DEVICE_STATE (* eDeviceState *)
VAR_OUTPUT
	(*if true, diagnosis info can be read by calling GetDeviceDiagnosisInfo*)
	xDiagnosisInfoAvailable	: BOOL;
	eError	: DED.ERROR;
END_VAR
//base implementation reads connector flags and delivers the right state
GetDeviceState := _diag.GetState(xDiagnosisInfoAvailable => xDiagnosisInfoAvailable, eError => eError);

//Sometimes you want to overload the connector flags state. Then use additionaly the following code.
IF GetDeviceState <> DED.DEVICE_STATE.DISABLED THEN
	IF GetBusState() = DED.BUS_STATE.ERROR THEN
		GetDeviceState := DED.DEVICE_STATE.ERROR;
	ELSE
		//TODO: return specific state
	END_IF
END_IF
END_METHOD

(* Returns true if the driver in the current state supports the requested communications state
 The method CheckSupportedCommunicationState is used to check for the general availability of communications states
 Therefore the result of CheckCurrentSupportedCommunicationState and CheckSupportedCommunicationState could differ if the driver is for example in the startup procedure and
 not supporting currently some communication states.*)
METHOD CheckCurrentSupportedCommunicationState : BOOL (* True, if state is supported*)
VAR_INPUT
	(* The communication state to check *)
	eRequestedState	: DED.DEVICE_TRANSITION_STATE;
END_VAR
CheckCurrentSupportedCommunicationState := (GetDeviceState() <> DED.DEVICE_STATE.DISABLED) AND CheckSupportedCommunicationState(eRequestedState);
END_METHOD

(* The implementation of this method returns true if the driver supports the requested communications state
 The application could query a driver to check if it is supporting specific communications states generally.
 The method CheckCurrentSupportedCommunicationState is used to check for the current state.
 Therefore the result of CheckCurrentSupportedCommunicationState and CheckSupportedCommunicationState could differ if the driver is for example in the startup procedure and
 not supporting currently some communication states.*)
METHOD CheckSupportedCommunicationState : BOOL (* True, if state is supported*)
VAR_INPUT
	(* The communication state to check *)
	eRequestedState	: DED.DEVICE_TRANSITION_STATE;
END_VAR
CASE eRequestedState OF
	DED.DEVICE_TRANSITION_STATE.RESET, DED.DEVICE_TRANSITION_STATE.START, DED.DEVICE_TRANSITION_STATE.STOP:
		CheckSupportedCommunicationState := TRUE;
END_CASE
END_METHOD

METHOD GetQoS : DED.ERROR
VAR_IN_OUT
	QualityInfo	: DED.QOS_INFO;
END_VAR
//TODO: Return quality of service informations e.g. busload, error counter,...
GetQoS := DED.ERROR.NOT_SUPPORTED;
END_METHOD

{attribute 'hide'}
(*Returns the bus error of the current node; you can also use functionblock GetBusError.*)
METHOD GetBusErrorAsync : DED.PROC_STATE (* eState *)
VAR_INPUT
	(*eCommand*)
	eCmd : DED.PROC_CMD;
END_VAR
VAR_IN_OUT
	(*error struct*)
	eriBusError	: DED.ERROR_INFO;
END_VAR
VAR_OUTPUT
	eError	: DED.ERROR;
END_VAR
//optional method; base implementation returns NOT_SUPPORTED
GetBusErrorAsync := _diag.GetErrorAsync(eCmd := eCmd, eriError := eriBusError, eError => eError);
END_METHOD

(*Returns a DiagnosisInfo if xDiagnosisInfoAvailable of GetBusState was true.*)
METHOD GetBusDiagnosisInfo : DED.ERROR (* eError *)
VAR_INPUT
	(*Pointer to memory*)
	pData	: CAA.PVOID;
	(*Size of memory in bytes where pData is pointing to*)
	szSize	: CAA.SIZE;
END_VAR
VAR_OUTPUT
	(*Number of Bytes written to pData*)
	szCount	: CAA.SIZE;
END_VAR
//This is an optional method. Return bus specific diagnostic information
GetBusDiagnosisInfo := DED.ERROR.NOT_SUPPORTED;
END_METHOD

(*Returns the bus state of the current node; if device state is ERROR further information can be read by GetBusError*)
METHOD GetBusState : DED.BUS_STATE (* eBusState *)
VAR_OUTPUT
	(*if true, diagnosis info can be read by calling GetBusDiagnosisInfo*)
	xDiagnosisInfoAvailable	: BOOL;
	eError	: DED.ERROR;
END_VAR
//base implementation reads connector flags and delivers the right state
GetBusState := _diag.GetBusState(xDiagnosisInfoAvailable => xDiagnosisInfoAvailable, eError => eError);

//Sometimes you want to overload the connector flags state. Then use additionaly the following code.
IF GetBusState <> DED.BUS_STATE.DISABLED THEN //if not disabled
	//TODO: return specific bus state 
END_IF
END_METHOD

(*Returns the bus information of the current node*)
METHOD GetBusInfo : DED.ERROR (*eError*)
VAR_IN_OUT
	(*Bus information struct*)
	buiInfo	: DED.BUS_INFO;
END_VAR
//base implementation supports all 3S specific fieldbusses.
GetBusInfo := _diag.GetBusInfo(buiInfo);
END_METHOD

(*Returns the fieldbus specific bus state; interpretation is fieldbus dependent*)
METHOD GetSpecificBusState : DED.ERROR (* eError *)
VAR_INPUT
	(*Pointer to memory*)
	pData	: CAA.PVOID;
	(*Size of memory in bytes where pData is pointing to*)
	szSize	: CAA.SIZE;
END_VAR
VAR_OUTPUT
	(*Number of Bytes written to pData*)
	szCount	: CAA.SIZE;
END_VAR
GetSpecificBusState := DED.ERROR.NOT_SUPPORTED;
END_METHOD

METHOD GetLogger : DED.ILogger
VAR_OUTPUT
	eError	: DED.ERROR;
END_VAR
eError := DED.ERROR.NOT_SUPPORTED;
END_METHOD

{attribute '''NORMAL__COMMENT' := 'Returns the bus scan of the current node'}
(*Returns the bus scan of the current node*)
METHOD GetBusScanAsync : DED.PROC_STATE
VAR_INPUT
	(*eCommand*)
	eCmd	: DED.PROC_CMD;
END_VAR
VAR_OUTPUT
	(* First node of scanned device list*)
	itfFirstDevice	: DED.INode;
	eError	: DED.ERROR;
END_VAR
//optional method; base implementation returns NOT_SUPPORTED
GetBusScanAsync := _diag.GetBusScanAsync(eCmd);
END_METHOD

(* This property is TRUE if reconfiguration is currently active.*)
{attribute 'conditionalshow' := '3SLib_Developer'}
PROPERTY ReconfigureActive : BOOL
GET
ReconfigureActive := _reconfig.ReconfigureActive;
END_GET
END_PROPERTY

(* Gets and sets the next sibling IReconfigureProvider.*)
{attribute 'conditionalshow' := '3SLib_Developer'}
PROPERTY SiblingIRP : DED.IReconfigureProvider
GET
SiblingIRP := _reconfig.SiblingIRP;
END_GET
SET
_reconfig.SiblingIRP := SiblingIRP;
END_SET
END_PROPERTY

(* Reconfigure reads the configuration of the corresponding node and applies it.
 Afterwards it calls ReconfigureAsync for all child IReconfigureProvider.
 After Reconfiguring all changed configuration values (Enable flag, Parameter changes,...) take effect.
 If the node doesn't support reconfiguring, method returns ERROR and eError contains |ERROR.NOT_SUPPORTED|.*)
 {attribute 'conditionalshow' := '3SLib_Developer'}
METHOD ReconfigureAsync : DED.PROC_STATE
VAR_INPUT
	(*eCommand: EXECUTE to start operation.*)
	eCmd	: DED.PROC_CMD;
	(*Originator of reconfiguration. 0 or current node if this is the first reconfiguration call.*)
	itfSender	: DED.INode;
END_VAR
VAR_OUTPUT
	(*Error code*)
	eError	: DED.ERROR;
END_VAR
//This method is used by CAA Device Diagnosis Reconfigure function block.
//The following example uses the reconfigure base implementation for I/O drivers. First it calls _reconfig.ReconfigureIoDriverAsync which uses IoStandard.IoMgrReconfigure.
//IoMgrReconfigure triggers a complete asynchronous reinitialization of the corresponding I/O driver 
//(IoDrvUpdateConfiguration with 0, IoDrvUpdatConfiguration with connectorlist and IoDrvUpdateMapping).
//Afterwards _reconfig.ReconfigureChildrenAsync is called which does a reconfigure on all children implementing IReconfigurationProvider. 
//For this it's necessary that _reconfig.Initialize_Diag is called in INode.Initialize_Diag!
//
//Note: It's also possible to implement Reconfigure in a different way e.g. if a stack supports Reconfigure for single child devices.
//In this case functionblocks for child devices have to implement IReconfigureProvider as well.

ReconfigureAsync := _reconfig.ReconfigureAsync(eCmd, itfSender, eError => eError);

(* CODE SNIPPET for custom specific implementation
{IF defined (pou:IoMgrReconfigure) AND defined (variable:ASYNCSTATE_READY)}
	CASE eCmd OF
		DED.PROC_CMD.EXECUTE:
			IF _byReconfigureState = 0 THEN
				IF itfSender = 0 THEN //if itfSender is current node ==> we are the originator; if someone calls us with 0, we also assume we are the originator.
					itfSender := THIS^; 
				END_IF
				
				_reconfig.BeginReconfigure(itfSender); //begin reconfiguration: if this is the first reconfigure call ==> enable flags are updated
				
				_xReconfigureError := FALSE; //member variable for memorizing errors
				_byReconfigureState := 1;
			END_IF
			
			IF _byReconfigureState = 1 THEN
				//TODO: Execute specific code
				//e.g. eProcState := ReconfigureNodeAsync(itfSender)
				IF eProcState = DED.PROC_STATE.DONE OR eProcState = DED.PROC_STATE.ERROR THEN
					_xReconfigureError := _xReconfigureError OR (eProcState = DED.PROC_STATE.ERROR);
					_byReconfigureState := 2;
				END_IF
			END_IF
			
			IF _byReconfigureState = 2 THEN
				//delegate reconfigure to all children implementing IReconfigureProvider (children are registered in Initialize_Diag by base implementation)
				eProcState := ReconfigureChildrenAsync(eCmd, itfSender);
				IF eProcState = DED.PROC_STATE.DONE OR eProcState = DED.PROC_STATE.ERROR THEN
					_xReconfigureError := _xReconfigureError OR (eProcState = DED.PROC_STATE.ERROR);
					_byReconfigureState := 0;
				END_IF
			END_IF

			IF _byReconfigureState <> 0 THEN
				ReconfigureAsync := DED.PROC_STATE.BUSY;
			ELSE
				IF _xReconfigureError THEN
					ReconfigureAsync := DED.PROC_STATE.ERROR;
					eError := DED.ERROR.ERROR_IO;
				ELSE
					ReconfigureAsync := DED.PROC_STATE.DONE;
				END_IF
				
				_reconfig.EndReconfigure(itfSender); //end reconfiguration
			END_IF
		ELSE
			//unexpected eCmd
			eError := DED.ERROR.PARAM_INVALID;
			ReconfigureAsync := DED.PROC_STATE.ERROR;
END_CASE
{ELSE}
	//old IoStandard library ==> reconfigure not supported
	ReconfigureAsync := DED.PROC_STATE.ERROR;
	eError := DED.ERROR.NOT_SUPPORTED;
{END_IF}
*)
END_METHOD

(* This method is used by IReconfigureProvider children to register at their parent.*)
{attribute 'conditionalshow' := '3SLib_Developer'}
METHOD RegisterIRPChild : DED.ERROR
VAR_INPUT
	itfChild	: DED.IReconfigureProvider;
END_VAR
RegisterIRPChild := _reconfig.RegisterIRPChild(itfChild);
END_METHOD

END_FUNCTION_BLOCK

// IoDrvMasterTemplateIEC/Function Blocks/IoDrvTemplateSlaveDiag
//This function block implements the diagnosis code for CAA Device Diagnosis.
{attribute 'no_assign'}
{attribute 'conditionalshow_all_locals' := 'IoDrvDebug'}
FUNCTION_BLOCK IoDrvTemplateSlaveDiag EXTENDS IoDrvTemplateSlave IMPLEMENTS DED.IDevice2 
VAR_INPUT
END_VAR
VAR_OUTPUT
END_VAR
VAR
	_diag : DED.CAADiagnosisBase;
	_tree : DED.CAADiagTreeBase;
END_VAR

(*Returns the number of childs below the current node*)
PROPERTY ChildNodeCount : CAA.COUNT
GET
ChildNodeCount := _tree.ChildNodeCount;
END_GET
END_PROPERTY

PROPERTY Connector : POINTER TO IoStandard.IoConfigConnector
GET
Connector := _tree.Connector;
END_GET
END_PROPERTY

(*This property returns if the node is enabled in the device tree. The setter can be used to change the Enabled flag. If enabling/disabling is not supported on the node the flag’s value will not change.*)
PROPERTY Enable : BOOL
GET
Enable := _tree.Enable;
END_GET
SET
_tree.Enable := Enable;
END_SET
END_PROPERTY

(*Returns the first child node below the current one*)
PROPERTY FirstChildNode : DED.INode
GET
FirstChildNode := _tree.FirstChildNode;
END_GET
END_PROPERTY

PROPERTY Index : UDINT
GET
Index := _tree.Index;
END_GET
SET
_tree.Index := Index;
END_SET
END_PROPERTY

(* returns true, if the current node is the root (plc) node, otherwise false*)
PROPERTY IsRootNode : BOOL
GET
IsRootNode := _tree.IsRootNode;
END_GET
END_PROPERTY

(* returns the next sibling node at the same level
 used for step through all nodes*)
PROPERTY NextSiblingNode : DED.INode
GET
NextSiblingNode := _tree.NextSiblingNode;
END_GET
END_PROPERTY

(* Returns the parent node or zero if already the root node is reached*)
PROPERTY ParentNode : DED.INode
GET
ParentNode := _tree.ParentNode;
END_GET
END_PROPERTY

(* Returns the number of sibling (same level) nodes*)
PROPERTY SiblingNodeCount : CAA.COUNT
GET
SiblingNodeCount := _tree.SiblingNodeCount;
END_GET
END_PROPERTY

{attribute 'hide'}
METHOD GetChild : DED.INode
VAR_INPUT
	udiIndex	: UDINT;
END_VAR
GetChild:= _tree.GetChild(udiIndex);
END_METHOD

{attribute 'hide'}
METHOD Initialize_Diag : UDINT
VAR_INPUT
	pConnector	: POINTER TO IoStandard.IoConfigConnector;
	nConnectorCount	: DINT;
	parent	: POINTER TO DED.INode;
	children	: POINTER TO DED.INode;
	udiChildCount	: UDINT;
END_VAR
//general initialization code: do not remove!
_tree.Initialize_Diag(pConnector, nConnectorCount, parent, children, udiChildCount);
_diag.Initialize_Diag(pConnector, nConnectorCount);

//if IReconfigureProvider is implemented
//_reconfig.Initialize_Diag(THIS^);
END_METHOD

{attribute '''NORMAL__COMMENT' := 'Returns the fieldbus specific device state; interpretation is fieldbus dependent'}
(*Returns the fieldbus specific device state; interpretation is fieldbus dependent*)
METHOD GetSpecificDeviceState : DED.ERROR (* eError *)
VAR_INPUT
	(*Pointer to memory*)
	pData	: CAA.PVOID;
	(*Size of memory in bytes where pData is pointing to*)
	szSize	: CAA.SIZE;
END_VAR
VAR_OUTPUT
	(*Number of Bytes written to pData*)
	szCount	: CAA.SIZE;
END_VAR
GetSpecificDeviceState := DED.ERROR.NOT_SUPPORTED;
END_METHOD

(*Starts, stops or resets a device*)
METHOD SetCommunicationState : DED.ERROR (* eError *)
VAR_INPUT
	eRequestedState	: DED.DEVICE_TRANSITION_STATE;
END_VAR
IF CheckCurrentSupportedCommunicationState(eRequestedState) THEN
	CASE eRequestedState OF
		DED.DEVICE_TRANSITION_STATE.RESET:
			//TODO: Send a reset command to the device.
		DED.DEVICE_TRANSITION_STATE.START:
			//TODO: Send a start command to the device.
		DED.DEVICE_TRANSITION_STATE.STOP:
			//TODO: Send a stop command to the device.
	END_CASE
ELSE
	SetCommunicationState := DED.ERROR.OPERATION_INVALID;
END_IF
END_METHOD

(*Returns the device information of the current node*)
METHOD GetDeviceInfo : DED.ERROR (*eError*)
VAR_IN_OUT
	(*Device information struct*)
	deiInfo	: DED.DEVICE_INFO;
END_VAR
//base implementation supports all 3S specific fieldbusses.
GetDeviceInfo := _diag.GetDeviceInfo(deiInfo);
END_METHOD

{attribute 'hide'}
(* Returns the device error of the current node; you can also use functionblock GetDeviceError.*)
METHOD GetDeviceErrorAsync : DED.PROC_STATE (* eState *)
VAR_INPUT
	(*eCommand*)
	eCmd	: DED.PROC_CMD;
END_VAR
VAR_IN_OUT
	(*error struct*)
	eriDeviceError	: DED.ERROR_INFO;
END_VAR
VAR_OUTPUT
	(*error code if method fails*)
	eError	: DED.ERROR;
END_VAR
//optional method; base implementation returns NOT_SUPPORTED
GetDeviceErrorAsync := _diag.GetErrorAsync(eCmd, eriDeviceError, eError => eError);
END_METHOD

{attribute 'hide'}
(*Returns the specific device error of the current node; interpretation is fieldbus-dependent; you can also use functionblock GetSpecificDeviceError*)
METHOD GetSpecificDeviceErrorAsync : DED.PROC_STATE (* eState *)
VAR_INPUT
	(*eCommand*)
	eCmd	: DED.PROC_CMD;
	(*Pointer to memory*)
	pData	: CAA.PVOID;
	(*Size of memory in bytes where pData is pointing to*)
	szSize	: CAA.SIZE;
END_VAR
VAR_OUTPUT
	(*Number of Bytes written to pData*)
	szCount	: CAA.SIZE;
	(*error code if method fails*)
	eError	: DED.ERROR;
END_VAR
//optional method; base implementation returns NOT_SUPPORTED
GetSpecificDeviceErrorAsync := _diag.GetSpecificDeviceErrorAsync(eCmd,pData, szSize, szCount=>szCount, eError => eError);
END_METHOD

{attribute '''NORMAL__COMMENT' := 'Returns a DiagnosisInfo if xDiagnosisInfoAvailable of GetDeviceState was true.'}
(*Returns a DiagnosisInfo if xDiagnosisInfoAvailable of GetDeviceState was true.*)
METHOD GetDeviceDiagnosisInfo : DED.ERROR (*eError*)
VAR_INPUT
	(*Pointer to memory*)
	pData	: CAA.PVOID;
	(*Size of memory in bytes where pData is pointing to*)
	szSize	: CAA.SIZE;
END_VAR
VAR_OUTPUT
	(*Number of Bytes written to pData*)
	szCount	: CAA.SIZE;
END_VAR
//This is an optional method. Return device specific diagnostic information
GetDeviceDiagnosisInfo := DED.ERROR.NOT_SUPPORTED;
END_METHOD

(*Returns the state of the device; if device state is ERROR further information can be read by GetDeviceError*)
METHOD GetDeviceState : DED.DEVICE_STATE (* eDeviceState *)
VAR_OUTPUT
	(*if true, diagnosis info can be read by calling GetDeviceDiagnosisInfo*)
	xDiagnosisInfoAvailable	: BOOL;
	eError	: DED.ERROR;
END_VAR
//base implementation reads connector flags and delivers the right state
GetDeviceState := _diag.GetState(xDiagnosisInfoAvailable => xDiagnosisInfoAvailable, eError => eError);

//Sometimes you want to overload the connector flags state. Then use additionaly the following code.
IF GetDeviceState <> DED.DEVICE_STATE.DISABLED THEN
	IF GetBusState() = DED.BUS_STATE.ERROR THEN
		GetDeviceState := DED.DEVICE_STATE.ERROR;
	ELSE
		//TODO: return specific state
	END_IF
END_IF
END_METHOD

(* Returns true if the driver in the current state supports the requested communications state
 The method CheckSupportedCommunicationState is used to check for the general availability of communications states
 Therefore the result of CheckCurrentSupportedCommunicationState and CheckSupportedCommunicationState could differ if the driver is for example in the startup procedure and
 not supporting currently some communication states.*)
METHOD CheckCurrentSupportedCommunicationState : BOOL (* True, if state is supported*)
VAR_INPUT
	(* The communication state to check *)
	eRequestedState	: DED.DEVICE_TRANSITION_STATE;
END_VAR
CheckCurrentSupportedCommunicationState := (GetDeviceState() <> DED.DEVICE_STATE.DISABLED) AND CheckSupportedCommunicationState(eRequestedState);
END_METHOD

(* The implementation of this method returns true if the driver supports the requested communications state
 The application could query a driver to check if it is supporting specific communications states generally.
 The method CheckCurrentSupportedCommunicationState is used to check for the current state.
 Therefore the result of CheckCurrentSupportedCommunicationState and CheckSupportedCommunicationState could differ if the driver is for example in the startup procedure and
 not supporting currently some communication states.*)
METHOD CheckSupportedCommunicationState : BOOL (* True, if state is supported*)
VAR_INPUT
	(* The communication state to check *)
	eRequestedState	: DED.DEVICE_TRANSITION_STATE;
END_VAR
CASE eRequestedState OF
	DED.DEVICE_TRANSITION_STATE.RESET, DED.DEVICE_TRANSITION_STATE.START, DED.DEVICE_TRANSITION_STATE.STOP:
		CheckSupportedCommunicationState := TRUE;
END_CASE
END_METHOD

METHOD GetQoS : DED.ERROR
VAR_IN_OUT
	QualityInfo	: DED.QOS_INFO;
END_VAR
//TODO: Return quality of service informations e.g. busload, error counter,...
GetQoS := DED.ERROR.NOT_SUPPORTED;
END_METHOD

{attribute 'hide'}
(*Returns the bus error of the current node; you can also use functionblock GetBusError.*)
METHOD GetBusErrorAsync : DED.PROC_STATE (* eState *)
VAR_INPUT
	(*eCommand*)
	eCmd : DED.PROC_CMD;
END_VAR
VAR_IN_OUT
	(*error struct*)
	eriBusError	: DED.ERROR_INFO;
END_VAR
VAR_OUTPUT
	eError	: DED.ERROR;
END_VAR
//optional method; base implementation returns NOT_SUPPORTED
GetBusErrorAsync := _diag.GetErrorAsync(eCmd := eCmd, eriError := eriBusError, eError => eError);
END_METHOD

(*Returns a DiagnosisInfo if xDiagnosisInfoAvailable of GetBusState was true.*)
METHOD GetBusDiagnosisInfo : DED.ERROR (* eError *)
VAR_INPUT
	(*Pointer to memory*)
	pData	: CAA.PVOID;
	(*Size of memory in bytes where pData is pointing to*)
	szSize	: CAA.SIZE;
END_VAR
VAR_OUTPUT
	(*Number of Bytes written to pData*)
	szCount	: CAA.SIZE;
END_VAR
//This is an optional method. Return bus specific diagnostic information
GetBusDiagnosisInfo := DED.ERROR.NOT_SUPPORTED;
END_METHOD

(*Returns the bus state of the current node; if device state is ERROR further information can be read by GetBusError*)
METHOD GetBusState : DED.BUS_STATE (* eBusState *)
VAR_OUTPUT
	(*if true, diagnosis info can be read by calling GetBusDiagnosisInfo*)
	xDiagnosisInfoAvailable	: BOOL;
	eError	: DED.ERROR;
END_VAR
//base implementation reads connector flags and delivers the right state
GetBusState := _diag.GetBusState(xDiagnosisInfoAvailable => xDiagnosisInfoAvailable, eError => eError);

//Sometimes you want to overload the connector flags state. Then use additionaly the following code.
IF GetBusState <> DED.BUS_STATE.DISABLED THEN //if not disabled
	//TODO: return specific bus state 
END_IF
END_METHOD

(*Returns the bus information of the current node*)
METHOD GetBusInfo : DED.ERROR (*eError*)
VAR_IN_OUT
	(*Bus information struct*)
	buiInfo	: DED.BUS_INFO;
END_VAR
//base implementation supports all 3S specific fieldbusses.
GetBusInfo := _diag.GetBusInfo(buiInfo);
END_METHOD

(*Returns the fieldbus specific bus state; interpretation is fieldbus dependent*)
METHOD GetSpecificBusState : DED.ERROR (* eError *)
VAR_INPUT
	(*Pointer to memory*)
	pData	: CAA.PVOID;
	(*Size of memory in bytes where pData is pointing to*)
	szSize	: CAA.SIZE;
END_VAR
VAR_OUTPUT
	(*Number of Bytes written to pData*)
	szCount	: CAA.SIZE;
END_VAR
GetSpecificBusState := DED.ERROR.NOT_SUPPORTED;
END_METHOD

END_FUNCTION_BLOCK

// IoDrvMasterTemplateIEC/Function Blocks/IoDrvTemplateModuleDiag
//This function block implements the diagnosis code for CAA Device Diagnosis.
{attribute 'no_assign'}
{attribute 'conditionalshow_all_locals' := 'IoDrvDebug'}
FUNCTION_BLOCK IoDrvTemplateModuleDiag EXTENDS IoDrvTemplateModule IMPLEMENTS DED.IDevice2
VAR_INPUT
END_VAR
VAR_OUTPUT
END_VAR
VAR
	_diag : DED.CAADiagnosisBase;
	_tree : DED.CAADiagTreeBase;
END_VAR

(*Returns the number of childs below the current node*)
PROPERTY ChildNodeCount : CAA.COUNT
GET
ChildNodeCount := _tree.ChildNodeCount;
END_GET
END_PROPERTY

PROPERTY Connector : POINTER TO IoStandard.IoConfigConnector
GET
Connector := _tree.Connector;
END_GET
END_PROPERTY

(*This property returns if the node is enabled in the device tree. The setter can be used to change the Enabled flag. If enabling/disabling is not supported on the node the flag’s value will not change.*)
PROPERTY Enable : BOOL
GET
Enable := _tree.Enable;
END_GET
SET
_tree.Enable := Enable;
END_SET
END_PROPERTY

(*Returns the first child node below the current one*)
PROPERTY FirstChildNode : DED.INode
GET
FirstChildNode := _tree.FirstChildNode;
END_GET
END_PROPERTY

PROPERTY Index : UDINT
GET
Index := _tree.Index;
END_GET
SET
_tree.Index := Index;
END_SET
END_PROPERTY

(* returns true, if the current node is the root (plc) node, otherwise false*)
PROPERTY IsRootNode : BOOL
GET
IsRootNode := _tree.IsRootNode;
END_GET
END_PROPERTY

(* returns the next sibling node at the same level
 used for step through all nodes*)
PROPERTY NextSiblingNode : DED.INode
GET
NextSiblingNode := _tree.NextSiblingNode;
END_GET
END_PROPERTY

(* Returns the parent node or zero if already the root node is reached*)
PROPERTY ParentNode : DED.INode
GET
ParentNode := _tree.ParentNode;
END_GET
END_PROPERTY

(* Returns the number of sibling (same level) nodes*)
PROPERTY SiblingNodeCount : CAA.COUNT
GET
SiblingNodeCount := _tree.SiblingNodeCount;
END_GET
END_PROPERTY

{attribute 'hide'}
METHOD GetChild : DED.INode
VAR_INPUT
	udiIndex	: UDINT;
END_VAR
GetChild:= _tree.GetChild(udiIndex);
END_METHOD

{attribute 'hide'}
METHOD Initialize_Diag : UDINT
VAR_INPUT
	pConnector	: POINTER TO IoStandard.IoConfigConnector;
	nConnectorCount	: DINT;
	parent	: POINTER TO DED.INode;
	children	: POINTER TO DED.INode;
	udiChildCount	: UDINT;
END_VAR
//general initialization code: do not remove!
_tree.Initialize_Diag(pConnector, nConnectorCount, parent, children, udiChildCount);
_diag.Initialize_Diag(pConnector, nConnectorCount);

//if IReconfigureProvider is implemented

//_reconfig.Initialize_Diag(THIS^);
END_METHOD

{attribute '''NORMAL__COMMENT' := 'Returns the fieldbus specific device state; interpretation is fieldbus dependent'}
(*Returns the fieldbus specific device state; interpretation is fieldbus dependent*)
METHOD GetSpecificDeviceState : DED.ERROR (* eError *)
VAR_INPUT
	(*Pointer to memory*)
	pData	: CAA.PVOID;
	(*Size of memory in bytes where pData is pointing to*)
	szSize	: CAA.SIZE;
END_VAR
VAR_OUTPUT
	(*Number of Bytes written to pData*)
	szCount	: CAA.SIZE;
END_VAR
GetSpecificDeviceState := DED.ERROR.NOT_SUPPORTED;
END_METHOD

(*Starts, stops or resets a device*)
METHOD SetCommunicationState : DED.ERROR (* eError *)
VAR_INPUT
	eRequestedState	: DED.DEVICE_TRANSITION_STATE;
END_VAR
IF CheckCurrentSupportedCommunicationState(eRequestedState) THEN
	CASE eRequestedState OF
		DED.DEVICE_TRANSITION_STATE.RESET:
			//TODO: Send a reset command to the device.
		DED.DEVICE_TRANSITION_STATE.START:
			//TODO: Send a start command to the device.
		DED.DEVICE_TRANSITION_STATE.STOP:
			//TODO: Send a stop command to the device.
	END_CASE
ELSE
	SetCommunicationState := DED.ERROR.OPERATION_INVALID;
END_IF
END_METHOD

(*Returns the device information of the current node*)
METHOD GetDeviceInfo : DED.ERROR (*eError*)
VAR_IN_OUT
	(*Device information struct*)
	deiInfo	: DED.DEVICE_INFO;
END_VAR
//base implementation supports all 3S specific fieldbusses.
GetDeviceInfo := _diag.GetDeviceInfo(deiInfo);
END_METHOD

{attribute 'hide'}
(* Returns the device error of the current node; you can also use functionblock GetDeviceError.*)
METHOD GetDeviceErrorAsync : DED.PROC_STATE (* eState *)
VAR_INPUT
	(*eCommand*)
	eCmd	: DED.PROC_CMD;
END_VAR
VAR_IN_OUT
	(*error struct*)
	eriDeviceError	: DED.ERROR_INFO;
END_VAR
VAR_OUTPUT
	(*error code if method fails*)
	eError	: DED.ERROR;
END_VAR
//optional method; base implementation returns NOT_SUPPORTED
GetDeviceErrorAsync := _diag.GetErrorAsync(eCmd, eriDeviceError, eError => eError);
END_METHOD

{attribute 'hide'}
(*Returns the specific device error of the current node; interpretation is fieldbus-dependent; you can also use functionblock GetSpecificDeviceError*)
METHOD GetSpecificDeviceErrorAsync : DED.PROC_STATE (* eState *)
VAR_INPUT
	(*eCommand*)
	eCmd	: DED.PROC_CMD;
	(*Pointer to memory*)
	pData	: CAA.PVOID;
	(*Size of memory in bytes where pData is pointing to*)
	szSize	: CAA.SIZE;
END_VAR
VAR_OUTPUT
	(*Number of Bytes written to pData*)
	szCount	: CAA.SIZE;
	(*error code if method fails*)
	eError	: DED.ERROR;
END_VAR
//optional method; base implementation returns NOT_SUPPORTED
GetSpecificDeviceErrorAsync := _diag.GetSpecificDeviceErrorAsync(eCmd,pData, szSize, szCount=>szCount, eError => eError);
END_METHOD

{attribute '''NORMAL__COMMENT' := 'Returns a DiagnosisInfo if xDiagnosisInfoAvailable of GetDeviceState was true.'}
(*Returns a DiagnosisInfo if xDiagnosisInfoAvailable of GetDeviceState was true.*)
METHOD GetDeviceDiagnosisInfo : DED.ERROR (*eError*)
VAR_INPUT
	(*Pointer to memory*)
	pData	: CAA.PVOID;
	(*Size of memory in bytes where pData is pointing to*)
	szSize	: CAA.SIZE;
END_VAR
VAR_OUTPUT
	(*Number of Bytes written to pData*)
	szCount	: CAA.SIZE;
END_VAR
//This is an optional method. Return device specific diagnostic information
GetDeviceDiagnosisInfo := DED.ERROR.NOT_SUPPORTED;
END_METHOD

(*Returns the state of the device; if device state is ERROR further information can be read by GetDeviceError*)
METHOD GetDeviceState : DED.DEVICE_STATE (* eDeviceState *)
VAR_OUTPUT
	(*if true, diagnosis info can be read by calling GetDeviceDiagnosisInfo*)
	xDiagnosisInfoAvailable	: BOOL;
	eError	: DED.ERROR;
END_VAR
//base implementation reads connector flags and delivers the right state
GetDeviceState := _diag.GetState(xDiagnosisInfoAvailable => xDiagnosisInfoAvailable, eError => eError);

//Sometimes you want to overload the connector flags state. Then use additionaly the following code.
IF GetDeviceState <> DED.DEVICE_STATE.DISABLED THEN
	IF GetBusState() = DED.BUS_STATE.ERROR THEN
		GetDeviceState := DED.DEVICE_STATE.ERROR;
	ELSE
		//TODO: return specific state
	END_IF
END_IF
END_METHOD

(* Returns true if the driver in the current state supports the requested communications state
 The method CheckSupportedCommunicationState is used to check for the general availability of communications states
 Therefore the result of CheckCurrentSupportedCommunicationState and CheckSupportedCommunicationState could differ if the driver is for example in the startup procedure and
 not supporting currently some communication states.*)
METHOD CheckCurrentSupportedCommunicationState : BOOL (* True, if state is supported*)
VAR_INPUT
	(* The communication state to check *)
	eRequestedState	: DED.DEVICE_TRANSITION_STATE;
END_VAR
CheckCurrentSupportedCommunicationState := (GetDeviceState() <> DED.DEVICE_STATE.DISABLED) AND CheckSupportedCommunicationState(eRequestedState);
END_METHOD

(* The implementation of this method returns true if the driver supports the requested communications state
 The application could query a driver to check if it is supporting specific communications states generally.
 The method CheckCurrentSupportedCommunicationState is used to check for the current state.
 Therefore the result of CheckCurrentSupportedCommunicationState and CheckSupportedCommunicationState could differ if the driver is for example in the startup procedure and
 not supporting currently some communication states.*)
METHOD CheckSupportedCommunicationState : BOOL (* True, if state is supported*)
VAR_INPUT
	(* The communication state to check *)
	eRequestedState	: DED.DEVICE_TRANSITION_STATE;
END_VAR
CASE eRequestedState OF
	DED.DEVICE_TRANSITION_STATE.RESET, DED.DEVICE_TRANSITION_STATE.START, DED.DEVICE_TRANSITION_STATE.STOP:
		CheckSupportedCommunicationState := TRUE;
END_CASE
END_METHOD

METHOD GetQoS : DED.ERROR
VAR_IN_OUT
	QualityInfo	: DED.QOS_INFO;
END_VAR
//TODO: Return quality of service informations e.g. busload, error counter,...
GetQoS := DED.ERROR.NOT_SUPPORTED;
END_METHOD

{attribute 'hide'}
(*Returns the bus error of the current node; you can also use functionblock GetBusError.*)
METHOD GetBusErrorAsync : DED.PROC_STATE (* eState *)
VAR_INPUT
	(*eCommand*)
	eCmd : DED.PROC_CMD;
END_VAR
VAR_IN_OUT
	(*error struct*)
	eriBusError	: DED.ERROR_INFO;
END_VAR
VAR_OUTPUT
	eError	: DED.ERROR;
END_VAR
//optional method; base implementation returns NOT_SUPPORTED
GetBusErrorAsync := _diag.GetErrorAsync(eCmd := eCmd, eriError := eriBusError, eError => eError);
END_METHOD

(*Returns a DiagnosisInfo if xDiagnosisInfoAvailable of GetBusState was true.*)
METHOD GetBusDiagnosisInfo : DED.ERROR (* eError *)
VAR_INPUT
	(*Pointer to memory*)
	pData	: CAA.PVOID;
	(*Size of memory in bytes where pData is pointing to*)
	szSize	: CAA.SIZE;
END_VAR
VAR_OUTPUT
	(*Number of Bytes written to pData*)
	szCount	: CAA.SIZE;
END_VAR
//This is an optional method. Return bus specific diagnostic information
GetBusDiagnosisInfo := DED.ERROR.NOT_SUPPORTED;
END_METHOD

(*Returns the bus state of the current node; if device state is ERROR further information can be read by GetBusError*)
METHOD GetBusState : DED.BUS_STATE (* eBusState *)
VAR_OUTPUT
	(*if true, diagnosis info can be read by calling GetBusDiagnosisInfo*)
	xDiagnosisInfoAvailable	: BOOL;
	eError	: DED.ERROR;
END_VAR
//base implementation reads connector flags and delivers the right state
GetBusState := _diag.GetBusState(xDiagnosisInfoAvailable => xDiagnosisInfoAvailable, eError => eError);

//Sometimes you want to overload the connector flags state. Then use additionaly the following code.
IF GetBusState <> DED.BUS_STATE.DISABLED THEN //if not disabled
	//TODO: return specific bus state 
END_IF
END_METHOD

(*Returns the bus information of the current node*)
METHOD GetBusInfo : DED.ERROR (*eError*)
VAR_IN_OUT
	(*Bus information struct*)
	buiInfo	: DED.BUS_INFO;
END_VAR
//base implementation supports all 3S specific fieldbusses.
GetBusInfo := _diag.GetBusInfo(buiInfo);
END_METHOD

(*Returns the fieldbus specific bus state; interpretation is fieldbus dependent*)
METHOD GetSpecificBusState : DED.ERROR (* eError *)
VAR_INPUT
	(*Pointer to memory*)
	pData	: CAA.PVOID;
	(*Size of memory in bytes where pData is pointing to*)
	szSize	: CAA.SIZE;
END_VAR
VAR_OUTPUT
	(*Number of Bytes written to pData*)
	szCount	: CAA.SIZE;
END_VAR
GetSpecificBusState := DED.ERROR.NOT_SUPPORTED;
END_METHOD

END_FUNCTION_BLOCK
